//     PlcTask Inputs/G_IO.arDI[75]/Ch[12] <-> Module 1 (GL20-1600END)/1600END input-bit maping/Digital input CH2-bit4
//     PlcTask Inputs/G_IO.arDI[75]/Ch[13] <-> Module 1 (GL20-1600END)/1600END input-bit maping/Digital input CH2-bit5
//     PlcTask Inputs/G_IO.arDI[75]/Ch[14] <-> Module 1 (GL20-1600END)/1600END input-bit maping/Digital input CH2-bit6
//     PlcTask Inputs/G_IO.arDI[75]/Ch[15] <-> Module 1 (GL20-1600END)/1600END input-bit maping/Digital input CH2-bit7
//     PlcTask Inputs/G_IO.arDI[75]/Ch[1] <-> Module 1 (GL20-1600END)/1600END input-bit maping/Digital input CH1-bit1
//     PlcTask Inputs/G_IO.arDI[75]/Ch[2] <-> Module 1 (GL20-1600END)/1600END input-bit maping/Digital input CH1-bit2
//     PlcTask Inputs/G_IO.arDI[75]/Ch[3] <-> Module 1 (GL20-1600END)/1600END input-bit maping/Digital input CH1-bit3
//     PlcTask Inputs/G_IO.arDI[75]/Ch[4] <-> Module 1 (GL20-1600END)/1600END input-bit maping/Digital input CH1-bit4
//     PlcTask Inputs/G_IO.arDI[75]/Ch[5] <-> Module 1 (GL20-1600END)/1600END input-bit maping/Digital input CH1-bit5
//     PlcTask Inputs/G_IO.arDI[75]/Ch[6] <-> Module 1 (GL20-1600END)/1600END input-bit maping/Digital input CH1-bit6
//     PlcTask Inputs/G_IO.arDI[75]/Ch[7] <-> Module 1 (GL20-1600END)/1600END input-bit maping/Digital input CH1-bit7
//     PlcTask Inputs/G_IO.arDI[75]/Ch[8] <-> Module 1 (GL20-1600END)/1600END input-bit maping/Digital input CH2-bit0
//     PlcTask Inputs/G_IO.arDI[75]/Ch[9] <-> Module 1 (GL20-1600END)/1600END input-bit maping/Digital input CH2-bit1
//     PlcTask Outputs/G_IO.arDO[75]/Ch[0] <-> Module 2 (GL20-0016ETP)/0016ETP Output-bit maping/Digital output CH1-bit0
//     PlcTask Outputs/G_IO.arDO[75]/Ch[10] <-> Module 2 (GL20-0016ETP)/0016ETP Output-bit maping/Digital output CH2-bit2
//     PlcTask Outputs/G_IO.arDO[75]/Ch[11] <-> Module 2 (GL20-0016ETP)/0016ETP Output-bit maping/Digital output CH2-bit3
//     PlcTask Outputs/G_IO.arDO[75]/Ch[12] <-> Module 2 (GL20-0016ETP)/0016ETP Output-bit maping/Digital output CH2-bit4
//     PlcTask Outputs/G_IO.arDO[75]/Ch[13] <-> Module 2 (GL20-0016ETP)/0016ETP Output-bit maping/Digital output CH2-bit5
//     PlcTask Outputs/G_IO.arDO[75]/Ch[14] <-> Module 2 (GL20-0016ETP)/0016ETP Output-bit maping/Digital output CH2-bit6
//     PlcTask Outputs/G_IO.arDO[75]/Ch[15] <-> Module 2 (GL20-0016ETP)/0016ETP Output-bit maping/Digital output CH2-bit7
//     PlcTask Outputs/G_IO.arDO[75]/Ch[1] <-> Module 2 (GL20-0016ETP)/0016ETP Output-bit maping/Digital output CH1-bit1
//     PlcTask Outputs/G_IO.arDO[75]/Ch[2] <-> Module 2 (GL20-0016ETP)/0016ETP Output-bit maping/Digital output CH1-bit2
//     PlcTask Outputs/G_IO.arDO[75]/Ch[3] <-> Module 2 (GL20-0016ETP)/0016ETP Output-bit maping/Digital output CH1-bit3
//     PlcTask Outputs/G_IO.arDO[75]/Ch[4] <-> Module 2 (GL20-0016ETP)/0016ETP Output-bit maping/Digital output CH1-bit4
//     PlcTask Outputs/G_IO.arDO[75]/Ch[5] <-> Module 2 (GL20-0016ETP)/0016ETP Output-bit maping/Digital output CH1-bit5
//     PlcTask Outputs/G_IO.arDO[75]/Ch[6] <-> Module 2 (GL20-0016ETP)/0016ETP Output-bit maping/Digital output CH1-bit6
//     PlcTask Outputs/G_IO.arDO[75]/Ch[7] <-> Module 2 (GL20-0016ETP)/0016ETP Output-bit maping/Digital output CH1-bit7
//     PlcTask Outputs/G_IO.arDO[75]/Ch[8] <-> Module 2 (GL20-0016ETP)/0016ETP Output-bit maping/Digital output CH2-bit0
//     PlcTask Outputs/G_IO.arDO[75]/Ch[9] <-> Module 2 (GL20-0016ETP)/0016ETP Output-bit maping/Digital output CH2-bit1
//   kittingDeca/kittingDeca Instance <-> pm side/fr1_dio
//     PlcTask Inputs/G_IO.arDI[76]/Ch[0] <-> Module 1 (GL20-1600END)/1600END input-bit maping/Digital input CH1-bit0
//     PlcTask Inputs/G_IO.arDI[76]/Ch[10] <-> Module 1 (GL20-1600END)/1600END input-bit maping/Digital input CH2-bit2
//     PlcTask Inputs/G_IO.arDI[76]/Ch[11] <-> Module 1 (GL20-1600END)/1600END input-bit maping/Digital input CH2-bit3
//     PlcTask Inputs/G_IO.arDI[76]/Ch[12] <-> Module 1 (GL20-1600END)/1600END input-bit maping/Digital input CH2-bit4
//     PlcTask Inputs/G_IO.arDI[76]/Ch[13] <-> Module 1 (GL20-1600END)/1600END input-bit maping/Digital input CH2-bit5
//     PlcTask Inputs/G_IO.arDI[76]/Ch[14] <-> Module 1 (GL20-1600END)/1600END input-bit maping/Digital input CH2-bit6
//     PlcTask Inputs/G_IO.arDI[76]/Ch[15] <-> Module 1 (GL20-1600END)/1600END input-bit maping/Digital input CH2-bit7
//     PlcTask Inputs/G_IO.arDI[76]/Ch[1] <-> Module 1 (GL20-1600END)/1600END input-bit maping/Digital input CH1-bit1
//     PlcTask Inputs/G_IO.arDI[76]/Ch[2] <-> Module 1 (GL20-1600END)/1600END input-bit maping/Digital input CH1-bit2
//     PlcTask Inputs/G_IO.arDI[76]/Ch[3] <-> Module 1 (GL20-1600END)/1600END input-bit maping/Digital input CH1-bit3
//     PlcTask Inputs/G_IO.arDI[76]/Ch[4] <-> Module 1 (GL20-1600END)/1600END input-bit maping/Digital input CH1-bit4
//     PlcTask Inputs/G_IO.arDI[76]/Ch[5] <-> Module 1 (GL20-1600END)/1600END input-bit maping/Digital input CH1-bit5
//     PlcTask Inputs/G_IO.arDI[76]/Ch[6] <-> Module 1 (GL20-1600END)/1600END input-bit maping/Digital input CH1-bit6
//     PlcTask Inputs/G_IO.arDI[76]/Ch[7] <-> Module 1 (GL20-1600END)/1600END input-bit maping/Digital input CH1-bit7
//     PlcTask Inputs/G_IO.arDI[76]/Ch[8] <-> Module 1 (GL20-1600END)/1600END input-bit maping/Digital input CH2-bit0
//     PlcTask Inputs/G_IO.arDI[76]/Ch[9] <-> Module 1 (GL20-1600END)/1600END input-bit maping/Digital input CH2-bit1
//     PlcTask Outputs/G_IO.arDO[76]/Ch[0] <-> Module 2 (GL20-0016ETP)/0016ETP Output-bit maping/Digital output CH1-bit0
//     PlcTask Outputs/G_IO.arDO[76]/Ch[10] <-> Module 2 (GL20-0016ETP)/0016ETP Output-bit maping/Digital output CH2-bit2
//     PlcTask Outputs/G_IO.arDO[76]/Ch[11] <-> Module 2 (GL20-0016ETP)/0016ETP Output-bit maping/Digital output CH2-bit3
//     PlcTask Outputs/G_IO.arDO[76]/Ch[12] <-> Module 2 (GL20-0016ETP)/0016ETP Output-bit maping/Digital output CH2-bit4
//     PlcTask Outputs/G_IO.arDO[76]/Ch[13] <-> Module 2 (GL20-0016ETP)/0016ETP Output-bit maping/Digital output CH2-bit5
//     PlcTask Outputs/G_IO.arDO[76]/Ch[14] <-> Module 2 (GL20-0016ETP)/0016ETP Output-bit maping/Digital output CH2-bit6
//     PlcTask Outputs/G_IO.arDO[76]/Ch[15] <-> Module 2 (GL20-0016ETP)/0016ETP Output-bit maping/Digital output CH2-bit7
//     PlcTask Outputs/G_IO.arDO[76]/Ch[1] <-> Module 2 (GL20-0016ETP)/0016ETP Output-bit maping/Digital output CH1-bit1
//     PlcTask Outputs/G_IO.arDO[76]/Ch[2] <-> Module 2 (GL20-0016ETP)/0016ETP Output-bit maping/Digital output CH1-bit2
//     PlcTask Outputs/G_IO.arDO[76]/Ch[3] <-> Module 2 (GL20-0016ETP)/0016ETP Output-bit maping/Digital output CH1-bit3
//     PlcTask Outputs/G_IO.arDO[76]/Ch[4] <-> Module 2 (GL20-0016ETP)/0016ETP Output-bit maping/Digital output CH1-bit4
//     PlcTask Outputs/G_IO.arDO[76]/Ch[5] <-> Module 2 (GL20-0016ETP)/0016ETP Output-bit maping/Digital output CH1-bit5
//     PlcTask Outputs/G_IO.arDO[76]/Ch[6] <-> Module 2 (GL20-0016ETP)/0016ETP Output-bit maping/Digital output CH1-bit6
//     PlcTask Outputs/G_IO.arDO[76]/Ch[7] <-> Module 2 (GL20-0016ETP)/0016ETP Output-bit maping/Digital output CH1-bit7
//     PlcTask Outputs/G_IO.arDO[76]/Ch[8] <-> Module 2 (GL20-0016ETP)/0016ETP Output-bit maping/Digital output CH2-bit0
//     PlcTask Outputs/G_IO.arDO[76]/Ch[9] <-> Module 2 (GL20-0016ETP)/0016ETP Output-bit maping/Digital output CH2-bit1
//   kittingDeca/kittingDeca Instance <-> pm side/lb0_converter
//     PlcTask Inputs/GVL.lb[0].belt[0].fbconverter.running_freq <-> Axis#1 Iutputs/Axis1 Running frequency
//     PlcTask Inputs/GVL.lb[0].belt[1].fbconverter.running_freq <-> Axis#2 Iutputs/Axis2 Running frequency
//     PlcTask Inputs/GVL.lb[0].belt[2].fbconverter.running_freq <-> Axis#3 Iutputs/Axis3 Running frequency
//     PlcTask Inputs/GVL.lb[0].belt[0].fbconverter.status <-> Axis#1 Iutputs/Axis1 AC drive running status word 2
//     PlcTask Inputs/GVL.lb[0].belt[1].fbconverter.status <-> Axis#2 Iutputs/Axis2 AC drive running status word 2
//     PlcTask Inputs/GVL.lb[0].belt[2].fbconverter.status <-> Axis#3 Iutputs/Axis3 AC drive running status word 2
//     PlcTask Outputs/GVL.lb[0].belt[0].fbconverter.cmd <-> Axis#1 Outputs/Axis1 Communication control command
//     PlcTask Outputs/GVL.lb[0].belt[1].fbconverter.cmd <-> Axis#2 Outputs/Axis2 Communication control command
//     PlcTask Outputs/GVL.lb[0].belt[2].fbconverter.cmd <-> Axis#3 Outputs/Axis3 Communication control command
//     PlcTask Outputs/GVL.lb[0].belt[0].fbconverter.freq <-> Axis#1 Outputs/Axis1 Frequency set through communication
//     PlcTask Outputs/GVL.lb[0].belt[1].fbconverter.freq <-> Axis#2 Outputs/Axis2 Frequency set through communication
//     PlcTask Outputs/GVL.lb[0].belt[2].fbconverter.freq <-> Axis#3 Outputs/Axis3 Frequency set through communication
//   kittingDeca/kittingDeca Instance <-> pm side/lb0_dio
//     PlcTask Inputs/G_IO.arDI[87]/Ch[0] <-> Module 1 (GL20-1600END)/1600END input-bit maping/Digital input CH1-bit0
//     PlcTask Inputs/G_IO.arDI[87]/Ch[10] <-> Module 1 (GL20-1600END)/1600END input-bit maping/Digital input CH2-bit2
//     PlcTask Inputs/G_IO.arDI[87]/Ch[11] <-> Module 1 (GL20-1600END)/1600END input-bit maping/Digital input CH2-bit3
//     PlcTask Inputs/G_IO.arDI[87]/Ch[12] <-> Module 1 (GL20-1600END)/1600END input-bit maping/Digital input CH2-bit4
//     PlcTask Inputs/G_IO.arDI[87]/Ch[13] <-> Module 1 (GL20-1600END)/1600END input-bit maping/Digital input CH2-bit5
//     PlcTask Inputs/G_IO.arDI[87]/Ch[14] <-> Module 1 (GL20-1600END)/1600END input-bit maping/Digital input CH2-bit6
//     PlcTask Inputs/G_IO.arDI[87]/Ch[15] <-> Module 1 (GL20-1600END)/1600END input-bit maping/Digital input CH2-bit7
//     PlcTask Inputs/G_IO.arDI[87]/Ch[1] <-> Module 1 (GL20-1600END)/1600END input-bit maping/Digital input CH1-bit1
//     PlcTask Inputs/G_IO.arDI[87]/Ch[2] <-> Module 1 (GL20-1600END)/1600END input-bit maping/Digital input CH1-bit2
//     PlcTask Inputs/G_IO.arDI[87]/Ch[3] <-> Module 1 (GL20-1600END)/1600END input-bit maping/Digital input CH1-bit3
//     PlcTask Inputs/G_IO.arDI[87]/Ch[4] <-> Module 1 (GL20-1600END)/1600END input-bit maping/Digital input CH1-bit4
//     PlcTask Inputs/G_IO.arDI[87]/Ch[5] <-> Module 1 (GL20-1600END)/1600END input-bit maping/Digital input CH1-bit5
//     PlcTask Inputs/G_IO.arDI[87]/Ch[6] <-> Module 1 (GL20-1600END)/1600END input-bit maping/Digital input CH1-bit6
//     PlcTask Inputs/G_IO.arDI[87]/Ch[7] <-> Module 1 (GL20-1600END)/1600END input-bit maping/Digital input CH1-bit7
//     PlcTask Inputs/G_IO.arDI[87]/Ch[8] <-> Module 1 (GL20-1600END)/1600END input-bit maping/Digital input CH2-bit0
//     PlcTask Inputs/G_IO.arDI[87]/Ch[9] <-> Module 1 (GL20-1600END)/1600END input-bit maping/Digital input CH2-bit1
//     PlcTask Outputs/G_IO.arDO[87]/Ch[0] <-> Module 2 (GL20-0016ETP)/0016ETP Output-bit maping/Digital output CH1-bit0
//     PlcTask Outputs/G_IO.arDO[87]/Ch[10] <-> Module 2 (GL20-0016ETP)/0016ETP Output-bit maping/Digital output CH2-bit2
//     PlcTask Outputs/G_IO.arDO[87]/Ch[11] <-> Module 2 (GL20-0016ETP)/0016ETP Output-bit maping/Digital output CH2-bit3
//     PlcTask Outputs/G_IO.arDO[87]/Ch[12] <-> Module 2 (GL20-0016ETP)/0016ETP Output-bit maping/Digital output CH2-bit4
//     PlcTask Outputs/G_IO.arDO[87]/Ch[13] <-> Module 2 (GL20-0016ETP)/0016ETP Output-bit maping/Digital output CH2-bit5
//     PlcTask Outputs/G_IO.arDO[87]/Ch[14] <-> Module 2 (GL20-0016ETP)/0016ETP Output-bit maping/Digital output CH2-bit6
//     PlcTask Outputs/G_IO.arDO[87]/Ch[15] <-> Module 2 (GL20-0016ETP)/0016ETP Output-bit maping/Digital output CH2-bit7
//     PlcTask Outputs/G_IO.arDO[87]/Ch[1] <-> Module 2 (GL20-0016ETP)/0016ETP Output-bit maping/Digital output CH1-bit1
//     PlcTask Outputs/G_IO.arDO[87]/Ch[2] <-> Module 2 (GL20-0016ETP)/0016ETP Output-bit maping/Digital output CH1-bit2
//     PlcTask Outputs/G_IO.arDO[87]/Ch[3] <-> Module 2 (GL20-0016ETP)/0016ETP Output-bit maping/Digital output CH1-bit3
//     PlcTask Outputs/G_IO.arDO[87]/Ch[4] <-> Module 2 (GL20-0016ETP)/0016ETP Output-bit maping/Digital output CH1-bit4
//     PlcTask Outputs/G_IO.arDO[87]/Ch[5] <-> Module 2 (GL20-0016ETP)/0016ETP Output-bit maping/Digital output CH1-bit5
//     PlcTask Outputs/G_IO.arDO[87]/Ch[6] <-> Module 2 (GL20-0016ETP)/0016ETP Output-bit maping/Digital output CH1-bit6
//     PlcTask Outputs/G_IO.arDO[87]/Ch[7] <-> Module 2 (GL20-0016ETP)/0016ETP Output-bit maping/Digital output CH1-bit7
//     PlcTask Outputs/G_IO.arDO[87]/Ch[8] <-> Module 2 (GL20-0016ETP)/0016ETP Output-bit maping/Digital output CH2-bit0
//     PlcTask Outputs/G_IO.arDO[87]/Ch[9] <-> Module 2 (GL20-0016ETP)/0016ETP Output-bit maping/Digital output CH2-bit1
//   kittingDeca/kittingDeca Instance <-> pm side/lb1_converter
//     PlcTask Inputs/GVL.lb[1].belt[0].fbconverter.running_freq <-> Axis#1 Iutputs/Axis1 Running frequency
//     PlcTask Inputs/GVL.lb[1].belt[1].fbconverter.running_freq <-> Axis#2 Iutputs/Axis2 Running frequency
//     PlcTask Inputs/GVL.lb[1].belt[2].fbconverter.running_freq <-> Axis#3 Iutputs/Axis3 Running frequency
//     PlcTask Inputs/GVL.lb[1].belt[0].fbconverter.status <-> Axis#1 Iutputs/Axis1 AC drive running status word 2
//     PlcTask Inputs/GVL.lb[1].belt[1].fbconverter.status <-> Axis#2 Iutputs/Axis2 AC drive running status word 2
//     PlcTask Inputs/GVL.lb[1].belt[2].fbconverter.status <-> Axis#3 Iutputs/Axis3 AC drive running status word 2
//     PlcTask Outputs/GVL.lb[1].belt[0].fbconverter.cmd <-> Axis#1 Outputs/Axis1 Communication control command
//     PlcTask Outputs/GVL.lb[1].belt[1].fbconverter.cmd <-> Axis#2 Outputs/Axis2 Communication control command
//     PlcTask Outputs/GVL.lb[1].belt[2].fbconverter.cmd <-> Axis#3 Outputs/Axis3 Communication control command
//     PlcTask Outputs/GVL.lb[1].belt[0].fbconverter.freq <-> Axis#1 Outputs/Axis1 Frequency set through communication
//     PlcTask Outputs/GVL.lb[1].belt[1].fbconverter.freq <-> Axis#2 Outputs/Axis2 Frequency set through communication
//     PlcTask Outputs/GVL.lb[1].belt[2].fbconverter.freq <-> Axis#3 Outputs/Axis3 Frequency set through communication
//   kittingDeca/kittingDeca Instance <-> pm side/lb1_dio
//     PlcTask Inputs/G_IO.arDI[90]/Ch[0] <-> Module 1 (GL20-1600END)/1600END input-bit maping/Digital input CH1-bit0
//     PlcTask Inputs/G_IO.arDI[90]/Ch[10] <-> Module 1 (GL20-1600END)/1600END input-bit maping/Digital input CH2-bit2
//     PlcTask Inputs/G_IO.arDI[90]/Ch[11] <-> Module 1 (GL20-1600END)/1600END input-bit maping/Digital input CH2-bit3
//     PlcTask Inputs/G_IO.arDI[90]/Ch[12] <-> Module 1 (GL20-1600END)/1600END input-bit maping/Digital input CH2-bit4
//     PlcTask Inputs/G_IO.arDI[90]/Ch[13] <-> Module 1 (GL20-1600END)/1600END input-bit maping/Digital input CH2-bit5
//     PlcTask Inputs/G_IO.arDI[90]/Ch[14] <-> Module 1 (GL20-1600END)/1600END input-bit maping/Digital input CH2-bit6
//     PlcTask Inputs/G_IO.arDI[90]/Ch[15] <-> Module 1 (GL20-1600END)/1600END input-bit maping/Digital input CH2-bit7
//     PlcTask Inputs/G_IO.arDI[90]/Ch[1] <-> Module 1 (GL20-1600END)/1600END input-bit maping/Digital input CH1-bit1
//     PlcTask Inputs/G_IO.arDI[90]/Ch[2] <-> Module 1 (GL20-1600END)/1600END input-bit maping/Digital input CH1-bit2
//     PlcTask Inputs/G_IO.arDI[90]/Ch[3] <-> Module 1 (GL20-1600END)/1600END input-bit maping/Digital input CH1-bit3
//     PlcTask Inputs/G_IO.arDI[90]/Ch[4] <-> Module 1 (GL20-1600END)/1600END input-bit maping/Digital input CH1-bit4
//     PlcTask Inputs/G_IO.arDI[90]/Ch[5] <-> Module 1 (GL20-1600END)/1600END input-bit maping/Digital input CH1-bit5
//     PlcTask Inputs/G_IO.arDI[90]/Ch[6] <-> Module 1 (GL20-1600END)/1600END input-bit maping/Digital input CH1-bit6
//     PlcTask Inputs/G_IO.arDI[90]/Ch[7] <-> Module 1 (GL20-1600END)/1600END input-bit maping/Digital input CH1-bit7
//     PlcTask Inputs/G_IO.arDI[90]/Ch[8] <-> Module 1 (GL20-1600END)/1600END input-bit maping/Digital input CH2-bit0
//     PlcTask Inputs/G_IO.arDI[90]/Ch[9] <-> Module 1 (GL20-1600END)/1600END input-bit maping/Digital input CH2-bit1
//     PlcTask Outputs/G_IO.arDO[90]/Ch[0] <-> Module 2 (GL20-0016ETP)/0016ETP Output-bit maping/Digital output CH1-bit0
//     PlcTask Outputs/G_IO.arDO[90]/Ch[10] <-> Module 2 (GL20-0016ETP)/0016ETP Output-bit maping/Digital output CH2-bit2
//     PlcTask Outputs/G_IO.arDO[90]/Ch[11] <-> Module 2 (GL20-0016ETP)/0016ETP Output-bit maping/Digital output CH2-bit3
//     PlcTask Outputs/G_IO.arDO[90]/Ch[12] <-> Module 2 (GL20-0016ETP)/0016ETP Output-bit maping/Digital output CH2-bit4
//     PlcTask Outputs/G_IO.arDO[90]/Ch[13] <-> Module 2 (GL20-0016ETP)/0016ETP Output-bit maping/Digital output CH2-bit5
//     PlcTask Outputs/G_IO.arDO[90]/Ch[14] <-> Module 2 (GL20-0016ETP)/0016ETP Output-bit maping/Digital output CH2-bit6
//     PlcTask Outputs/G_IO.arDO[90]/Ch[15] <-> Module 2 (GL20-0016ETP)/0016ETP Output-bit maping/Digital output CH2-bit7
//     PlcTask Outputs/G_IO.arDO[90]/Ch[1] <-> Module 2 (GL20-0016ETP)/0016ETP Output-bit maping/Digital output CH1-bit1
//     PlcTask Outputs/G_IO.arDO[90]/Ch[2] <-> Module 2 (GL20-0016ETP)/0016ETP Output-bit maping/Digital output CH1-bit2
//     PlcTask Outputs/G_IO.arDO[90]/Ch[3] <-> Module 2 (GL20-0016ETP)/0016ETP Output-bit maping/Digital output CH1-bit3
//     PlcTask Outputs/G_IO.arDO[90]/Ch[4] <-> Module 2 (GL20-0016ETP)/0016ETP Output-bit maping/Digital output CH1-bit4
//     PlcTask Outputs/G_IO.arDO[90]/Ch[5] <-> Module 2 (GL20-0016ETP)/0016ETP Output-bit maping/Digital output CH1-bit5
//     PlcTask Outputs/G_IO.arDO[90]/Ch[6] <-> Module 2 (GL20-0016ETP)/0016ETP Output-bit maping/Digital output CH1-bit6
//     PlcTask Outputs/G_IO.arDO[90]/Ch[7] <-> Module 2 (GL20-0016ETP)/0016ETP Output-bit maping/Digital output CH1-bit7
//     PlcTask Outputs/G_IO.arDO[90]/Ch[8] <-> Module 2 (GL20-0016ETP)/0016ETP Output-bit maping/Digital output CH2-bit0
//     PlcTask Outputs/G_IO.arDO[90]/Ch[9] <-> Module 2 (GL20-0016ETP)/0016ETP Output-bit maping/Digital output CH2-bit1
//   kittingDeca/kittingDeca Instance <-> pm side/lc0_converter
//     PlcTask Inputs/GVL.lc[0].belt_out.belt.fbconverter.running_freq <-> Axis#1 Iutputs/Axis1 Running frequency
//     PlcTask Inputs/GVL.lc[0].belt_out.belt.fbconverter.status <-> Axis#1 Iutputs/Axis1 AC drive running status word 2
//     PlcTask Outputs/GVL.lc[0].belt_out.belt.fbconverter.cmd <-> Axis#1 Outputs/Axis1 Communication control command
//     PlcTask Outputs/GVL.lc[0].belt_out.belt.fbconverter.freq <-> Axis#1 Outputs/Axis1 Frequency set through communication
//   kittingDeca/kittingDeca Instance <-> pm side/lc0_dio
//     PlcTask Inputs/G_IO.arDI[85]/Ch[0] <-> Module 1 (GL20-1600END)/1600END input-bit maping/Digital input CH1-bit0
//     PlcTask Inputs/G_IO.arDI[85]/Ch[10] <-> Module 1 (GL20-1600END)/1600END input-bit maping/Digital input CH2-bit2
//     PlcTask Inputs/G_IO.arDI[85]/Ch[11] <-> Module 1 (GL20-1600END)/1600END input-bit maping/Digital input CH2-bit3
//     PlcTask Inputs/G_IO.arDI[85]/Ch[12] <-> Module 1 (GL20-1600END)/1600END input-bit maping/Digital input CH2-bit4
//     PlcTask Inputs/G_IO.arDI[85]/Ch[13] <-> Module 1 (GL20-1600END)/1600END input-bit maping/Digital input CH2-bit5
//     PlcTask Inputs/G_IO.arDI[85]/Ch[14] <-> Module 1 (GL20-1600END)/1600END input-bit maping/Digital input CH2-bit6
//     PlcTask Inputs/G_IO.arDI[85]/Ch[15] <-> Module 1 (GL20-1600END)/1600END input-bit maping/Digital input CH2-bit7
//     PlcTask Inputs/G_IO.arDI[85]/Ch[1] <-> Module 1 (GL20-1600END)/1600END input-bit maping/Digital input CH1-bit1
//     PlcTask Inputs/G_IO.arDI[85]/Ch[2] <-> Module 1 (GL20-1600END)/1600END input-bit maping/Digital input CH1-bit2
//     PlcTask Inputs/G_IO.arDI[85]/Ch[3] <-> Module 1 (GL20-1600END)/1600END input-bit maping/Digital input CH1-bit3
//     PlcTask Inputs/G_IO.arDI[85]/Ch[4] <-> Module 1 (GL20-1600END)/1600END input-bit maping/Digital input CH1-bit4
//     PlcTask Inputs/G_IO.arDI[85]/Ch[5] <-> Module 1 (GL20-1600END)/1600END input-bit maping/Digital input CH1-bit5
//     PlcTask Inputs/G_IO.arDI[85]/Ch[6] <-> Module 1 (GL20-1600END)/1600END input-bit maping/Digital input CH1-bit6
//     PlcTask Inputs/G_IO.arDI[85]/Ch[7] <-> Module 1 (GL20-1600END)/1600END input-bit maping/Digital input CH1-bit7
//     PlcTask Inputs/G_IO.arDI[85]/Ch[8] <-> Module 1 (GL20-1600END)/1600END input-bit maping/Digital input CH2-bit0
//     PlcTask Inputs/G_IO.arDI[85]/Ch[9] <-> Module 1 (GL20-1600END)/1600END input-bit maping/Digital input CH2-bit1
//     PlcTask Inputs/G_IO.arDI[86]/Ch[0] <-> Module 2 (GL20-1600END)/1600END input-bit maping/Digital input CH1-bit0
//     PlcTask Inputs/G_IO.arDI[86]/Ch[10] <-> Module 2 (GL20-1600END)/1600END input-bit maping/Digital input CH2-bit2
//     PlcTask Inputs/G_IO.arDI[86]/Ch[11] <-> Module 2 (GL20-1600END)/1600END input-bit maping/Digital input CH2-bit3
//     PlcTask Inputs/G_IO.arDI[86]/Ch[12] <-> Module 2 (GL20-1600END)/1600END input-bit maping/Digital input CH2-bit4
//     PlcTask Inputs/G_IO.arDI[86]/Ch[13] <-> Module 2 (GL20-1600END)/1600END input-bit maping/Digital input CH2-bit5
//     PlcTask Inputs/G_IO.arDI[86]/Ch[14] <-> Module 2 (GL20-1600END)/1600END input-bit maping/Digital input CH2-bit6
//     PlcTask Inputs/G_IO.arDI[86]/Ch[15] <-> Module 2 (GL20-1600END)/1600END input-bit maping/Digital input CH2-bit7
//     PlcTask Inputs/G_IO.arDI[86]/Ch[1] <-> Module 2 (GL20-1600END)/1600END input-bit maping/Digital input CH1-bit1
//     PlcTask Inputs/G_IO.arDI[86]/Ch[2] <-> Module 2 (GL20-1600END)/1600END input-bit maping/Digital input CH1-bit2
//     PlcTask Inputs/G_IO.arDI[86]/Ch[3] <-> Module 2 (GL20-1600END)/1600END input-bit maping/Digital input CH1-bit3
//     PlcTask Inputs/G_IO.arDI[86]/Ch[4] <-> Module 2 (GL20-1600END)/1600END input-bit maping/Digital input CH1-bit4
//     PlcTask Inputs/G_IO.arDI[86]/Ch[5] <-> Module 2 (GL20-1600END)/1600END input-bit maping/Digital input CH1-bit5
//     PlcTask Inputs/G_IO.arDI[86]/Ch[6] <-> Module 2 (GL20-1600END)/1600END input-bit maping/Digital input CH1-bit6
//     PlcTask Inputs/G_IO.arDI[86]/Ch[7] <-> Module 2 (GL20-1600END)/1600END input-bit maping/Digital input CH1-bit7
//     PlcTask Inputs/G_IO.arDI[86]/Ch[8] <-> Module 2 (GL20-1600END)/1600END input-bit maping/Digital input CH2-bit0
//     PlcTask Inputs/G_IO.arDI[86]/Ch[9] <-> Module 2 (GL20-1600END)/1600END input-bit maping/Digital input CH2-bit1
//     PlcTask Outputs/G_IO.arDO[85]/Ch[0] <-> Module 3 (GL20-0016ETP)/0016ETP Output-bit maping/Digital output CH1-bit0
//     PlcTask Outputs/G_IO.arDO[85]/Ch[10] <-> Module 3 (GL20-0016ETP)/0016ETP Output-bit maping/Digital output CH2-bit2
//     PlcTask Outputs/G_IO.arDO[85]/Ch[11] <-> Module 3 (GL20-0016ETP)/0016ETP Output-bit maping/Digital output CH2-bit3
//     PlcTask Outputs/G_IO.arDO[85]/Ch[12] <-> Module 3 (GL20-0016ETP)/0016ETP Output-bit maping/Digital output CH2-bit4
//     PlcTask Outputs/G_IO.arDO[85]/Ch[13] <-> Module 3 (GL20-0016ETP)/0016ETP Output-bit maping/Digital output CH2-bit5
//     PlcTask Outputs/G_IO.arDO[85]/Ch[14] <-> Module 3 (GL20-0016ETP)/0016ETP Output-bit maping/Digital output CH2-bit6
//     PlcTask Outputs/G_IO.arDO[85]/Ch[15] <-> Module 3 (GL20-0016ETP)/0016ETP Output-bit maping/Digital output CH2-bit7
//     PlcTask Outputs/G_IO.arDO[85]/Ch[1] <-> Module 3 (GL20-0016ETP)/0016ETP Output-bit maping/Digital output CH1-bit1
//     PlcTask Outputs/G_IO.arDO[85]/Ch[2] <-> Module 3 (GL20-0016ETP)/0016ETP Output-bit maping/Digital output CH1-bit2
//     PlcTask Outputs/G_IO.arDO[85]/Ch[3] <-> Module 3 (GL20-0016ETP)/0016ETP Output-bit maping/Digital output CH1-bit3
//     PlcTask Outputs/G_IO.arDO[85]/Ch[4] <-> Module 3 (GL20-0016ETP)/0016ETP Output-bit maping/Digital output CH1-bit4
//     PlcTask Outputs/G_IO.arDO[85]/Ch[5] <-> Module 3 (GL20-0016ETP)/0016ETP Output-bit maping/Digital output CH1-bit5
//     PlcTask Outputs/G_IO.arDO[85]/Ch[6] <-> Module 3 (GL20-0016ETP)/0016ETP Output-bit maping/Digital output CH1-bit6
//     PlcTask Outputs/G_IO.arDO[85]/Ch[7] <-> Module 3 (GL20-0016ETP)/0016ETP Output-bit maping/Digital output CH1-bit7
//     PlcTask Outputs/G_IO.arDO[85]/Ch[8] <-> Module 3 (GL20-0016ETP)/0016ETP Output-bit maping/Digital output CH2-bit0
//     PlcTask Outputs/G_IO.arDO[85]/Ch[9] <-> Module 3 (GL20-0016ETP)/0016ETP Output-bit maping/Digital output CH2-bit1
//     PlcTask Outputs/G_IO.arDO[86]/Ch[0] <-> Module 4 (GL20-0016ETP)/0016ETP Output-bit maping/Digital output CH1-bit0
//     PlcTask Outputs/G_IO.arDO[86]/Ch[10] <-> Module 4 (GL20-0016ETP)/0016ETP Output-bit maping/Digital output CH2-bit2
//     PlcTask Outputs/G_IO.arDO[86]/Ch[11] <-> Module 4 (GL20-0016ETP)/0016ETP Output-bit maping/Digital output CH2-bit3
//     PlcTask Outputs/G_IO.arDO[86]/Ch[12] <-> Module 4 (GL20-0016ETP)/0016ETP Output-bit maping/Digital output CH2-bit4
//     PlcTask Outputs/G_IO.arDO[86]/Ch[13] <-> Module 4 (GL20-0016ETP)/0016ETP Output-bit maping/Digital output CH2-bit5
//     PlcTask Outputs/G_IO.arDO[86]/Ch[14] <-> Module 4 (GL20-0016ETP)/0016ETP Output-bit maping/Digital output CH2-bit6
//     PlcTask Outputs/G_IO.arDO[86]/Ch[15] <-> Module 4 (GL20-0016ETP)/0016ETP Output-bit maping/Digital output CH2-bit7
//     PlcTask Outputs/G_IO.arDO[86]/Ch[1] <-> Module 4 (GL20-0016ETP)/0016ETP Output-bit maping/Digital output CH1-bit1
//     PlcTask Outputs/G_IO.arDO[86]/Ch[2] <-> Module 4 (GL20-0016ETP)/0016ETP Output-bit maping/Digital output CH1-bit2
//     PlcTask Outputs/G_IO.arDO[86]/Ch[3] <-> Module 4 (GL20-0016ETP)/0016ETP Output-bit maping/Digital output CH1-bit3
//     PlcTask Outputs/G_IO.arDO[86]/Ch[4] <-> Module 4 (GL20-0016ETP)/0016ETP Output-bit maping/Digital output CH1-bit4
//     PlcTask Outputs/G_IO.arDO[86]/Ch[5] <-> Module 4 (GL20-0016ETP)/0016ETP Output-bit maping/Digital output CH1-bit5
//     PlcTask Outputs/G_IO.arDO[86]/Ch[6] <-> Module 4 (GL20-0016ETP)/0016ETP Output-bit maping/Digital output CH1-bit6
//     PlcTask Outputs/G_IO.arDO[86]/Ch[7] <-> Module 4 (GL20-0016ETP)/0016ETP Output-bit maping/Digital output CH1-bit7
//     PlcTask Outputs/G_IO.arDO[86]/Ch[8] <-> Module 4 (GL20-0016ETP)/0016ETP Output-bit maping/Digital output CH2-bit0
//     PlcTask Outputs/G_IO.arDO[86]/Ch[9] <-> Module 4 (GL20-0016ETP)/0016ETP Output-bit maping/Digital output CH2-bit1
//   kittingDeca/kittingDeca Instance <-> pm side/lc1_converter
//     PlcTask Inputs/GVL.lc[1].belt_out.belt.fbconverter.running_freq <-> Axis#1 Iutputs/Axis1 Running frequency
//     PlcTask Inputs/GVL.lc[1].belt_out.belt.fbconverter.status <-> Axis#1 Iutputs/Axis1 AC drive running status word 2
//     PlcTask Outputs/GVL.lc[1].belt_out.belt.fbconverter.cmd <-> Axis#1 Outputs/Axis1 Communication control command
//     PlcTask Outputs/GVL.lc[1].belt_out.belt.fbconverter.freq <-> Axis#1 Outputs/Axis1 Frequency set through communication
//   kittingDeca/kittingDeca Instance <-> pm side/lc1_dio
//     PlcTask Inputs/G_IO.arDI[88]/Ch[0] <-> Module 1 (GL20-1600END)/1600END input-bit maping/Digital input CH1-bit0
//     PlcTask Inputs/G_IO.arDI[88]/Ch[10] <-> Module 1 (GL20-1600END)/1600END input-bit maping/Digital input CH2-bit2
//     PlcTask Inputs/G_IO.arDI[88]/Ch[11] <-> Module 1 (GL20-1600END)/1600END input-bit maping/Digital input CH2-bit3
//     PlcTask Inputs/G_IO.arDI[88]/Ch[12] <-> Module 1 (GL20-1600END)/1600END input-bit maping/Digital input CH2-bit4
//     PlcTask Inputs/G_IO.arDI[88]/Ch[13] <-> Module 1 (GL20-1600END)/1600END input-bit maping/Digital input CH2-bit5
//     PlcTask Inputs/G_IO.arDI[88]/Ch[14] <-> Module 1 (GL20-1600END)/1600END input-bit maping/Digital input CH2-bit6
//     PlcTask Inputs/G_IO.arDI[88]/Ch[15] <-> Module 1 (GL20-1600END)/1600END input-bit maping/Digital input CH2-bit7
//     PlcTask Inputs/G_IO.arDI[88]/Ch[1] <-> Module 1 (GL20-1600END)/1600END input-bit maping/Digital input CH1-bit1
//     PlcTask Inputs/G_IO.arDI[88]/Ch[2] <-> Module 1 (GL20-1600END)/1600END input-bit maping/Digital input CH1-bit2
//     PlcTask Inputs/G_IO.arDI[88]/Ch[3] <-> Module 1 (GL20-1600END)/1600END input-bit maping/Digital input CH1-bit3
//     PlcTask Inputs/G_IO.arDI[88]/Ch[4] <-> Module 1 (GL20-1600END)/1600END input-bit maping/Digital input CH1-bit4
//     PlcTask Inputs/G_IO.arDI[88]/Ch[5] <-> Module 1 (GL20-1600END)/1600END input-bit maping/Digital input CH1-bit5
//     PlcTask Inputs/G_IO.arDI[88]/Ch[6] <-> Module 1 (GL20-1600END)/1600END input-bit maping/Digital input CH1-bit6
//     PlcTask Inputs/G_IO.arDI[88]/Ch[7] <-> Module 1 (GL20-1600END)/1600END input-bit maping/Digital input CH1-bit7
//     PlcTask Inputs/G_IO.arDI[88]/Ch[8] <-> Module 1 (GL20-1600END)/1600END input-bit maping/Digital input CH2-bit0
//     PlcTask Inputs/G_IO.arDI[88]/Ch[9] <-> Module 1 (GL20-1600END)/1600END input-bit maping/Digital input CH2-bit1
//     PlcTask Inputs/G_IO.arDI[89]/Ch[0] <-> Module 2 (GL20-1600END)/1600END input-bit maping/Digital input CH1-bit0
//     PlcTask Inputs/G_IO.arDI[89]/Ch[10] <-> Module 2 (GL20-1600END)/1600END input-bit maping/Digital input CH2-bit2
//     PlcTask Inputs/G_IO.arDI[89]/Ch[11] <-> Module 2 (GL20-1600END)/1600END input-bit maping/Digital input CH2-bit3
//     PlcTask Inputs/G_IO.arDI[89]/Ch[12] <-> Module 2 (GL20-1600END)/1600END input-bit maping/Digital input CH2-bit4
//     PlcTask Inputs/G_IO.arDI[89]/Ch[13] <-> Module 2 (GL20-1600END)/1600END input-bit maping/Digital input CH2-bit5
//     PlcTask Inputs/G_IO.arDI[89]/Ch[14] <-> Module 2 (GL20-1600END)/1600END input-bit maping/Digital input CH2-bit6
//     PlcTask Inputs/G_IO.arDI[89]/Ch[15] <-> Module 2 (GL20-1600END)/1600END input-bit maping/Digital input CH2-bit7
//     PlcTask Inputs/G_IO.arDI[89]/Ch[1] <-> Module 2 (GL20-1600END)/1600END input-bit maping/Digital input CH1-bit1
//     PlcTask Inputs/G_IO.arDI[89]/Ch[2] <-> Module 2 (GL20-1600END)/1600END input-bit maping/Digital input CH1-bit2
//     PlcTask Inputs/G_IO.arDI[89]/Ch[3] <-> Module 2 (GL20-1600END)/1600END input-bit maping/Digital input CH1-bit3
//     PlcTask Inputs/G_IO.arDI[89]/Ch[4] <-> Module 2 (GL20-1600END)/1600END input-bit maping/Digital input CH1-bit4
//     PlcTask Inputs/G_IO.arDI[89]/Ch[5] <-> Module 2 (GL20-1600END)/1600END input-bit maping/Digital input CH1-bit5
//     PlcTask Inputs/G_IO.arDI[89]/Ch[6] <-> Module 2 (GL20-1600END)/1600END input-bit maping/Digital input CH1-bit6
//     PlcTask Inputs/G_IO.arDI[89]/Ch[7] <-> Module 2 (GL20-1600END)/1600END input-bit maping/Digital input CH1-bit7
//     PlcTask Inputs/G_IO.arDI[89]/Ch[8] <-> Module 2 (GL20-1600END)/1600END input-bit maping/Digital input CH2-bit0
//     PlcTask Inputs/G_IO.arDI[89]/Ch[9] <-> Module 2 (GL20-1600END)/1600END input-bit maping/Digital input CH2-bit1
//     PlcTask Outputs/G_IO.arDO[88]/Ch[0] <-> Module 3 (GL20-0016ETP)/0016ETP Output-bit maping/Digital output CH1-bit0
//     PlcTask Outputs/G_IO.arDO[88]/Ch[10] <-> Module 3 (GL20-0016ETP)/0016ETP Output-bit maping/Digital output CH2-bit2
//     PlcTask Outputs/G_IO.arDO[88]/Ch[11] <-> Module 3 (GL20-0016ETP)/0016ETP Output-bit maping/Digital output CH2-bit3
//     PlcTask Outputs/G_IO.arDO[88]/Ch[12] <-> Module 3 (GL20-0016ETP)/0016ETP Output-bit maping/Digital output CH2-bit4
//     PlcTask Outputs/G_IO.arDO[88]/Ch[13] <-> Module 3 (GL20-0016ETP)/0016ETP Output-bit maping/Digital output CH2-bit5
//     PlcTask Outputs/G_IO.arDO[88]/Ch[14] <-> Module 3 (GL20-0016ETP)/0016ETP Output-bit maping/Digital output CH2-bit6
//     PlcTask Outputs/G_IO.arDO[88]/Ch[15] <-> Module 3 (GL20-0016ETP)/0016ETP Output-bit maping/Digital output CH2-bit7
//     PlcTask Outputs/G_IO.arDO[88]/Ch[1] <-> Module 3 (GL20-0016ETP)/0016ETP Output-bit maping/Digital output CH1-bit1
//     PlcTask Outputs/G_IO.arDO[88]/Ch[2] <-> Module 3 (GL20-0016ETP)/0016ETP Output-bit maping/Digital output CH1-bit2
//     PlcTask Outputs/G_IO.arDO[88]/Ch[3] <-> Module 3 (GL20-0016ETP)/0016ETP Output-bit maping/Digital output CH1-bit3
//     PlcTask Outputs/G_IO.arDO[88]/Ch[4] <-> Module 3 (GL20-0016ETP)/0016ETP Output-bit maping/Digital output CH1-bit4
//     PlcTask Outputs/G_IO.arDO[88]/Ch[5] <-> Module 3 (GL20-0016ETP)/0016ETP Output-bit maping/Digital output CH1-bit5
//     PlcTask Outputs/G_IO.arDO[88]/Ch[6] <-> Module 3 (GL20-0016ETP)/0016ETP Output-bit maping/Digital output CH1-bit6
//     PlcTask Outputs/G_IO.arDO[88]/Ch[7] <-> Module 3 (GL20-0016ETP)/0016ETP Output-bit maping/Digital output CH1-bit7
//     PlcTask Outputs/G_IO.arDO[88]/Ch[8] <-> Module 3 (GL20-0016ETP)/0016ETP Output-bit maping/Digital output CH2-bit0
//     PlcTask Outputs/G_IO.arDO[88]/Ch[9] <-> Module 3 (GL20-0016ETP)/0016ETP Output-bit maping/Digital output CH2-bit1
//     PlcTask Outputs/G_IO.arDO[89]/Ch[0] <-> Module 4 (GL20-0016ETP)/0016ETP Output-bit maping/Digital output CH1-bit0
//     PlcTask Outputs/G_IO.arDO[89]/Ch[10] <-> Module 4 (GL20-0016ETP)/0016ETP Output-bit maping/Digital output CH2-bit2
//     PlcTask Outputs/G_IO.arDO[89]/Ch[11] <-> Module 4 (GL20-0016ETP)/0016ETP Output-bit maping/Digital output CH2-bit3
//     PlcTask Outputs/G_IO.arDO[89]/Ch[12] <-> Module 4 (GL20-0016ETP)/0016ETP Output-bit maping/Digital output CH2-bit4
//     PlcTask Outputs/G_IO.arDO[89]/Ch[13] <-> Module 4 (GL20-0016ETP)/0016ETP Output-bit maping/Digital output CH2-bit5
//     PlcTask Outputs/G_IO.arDO[89]/Ch[14] <-> Module 4 (GL20-0016ETP)/0016ETP Output-bit maping/Digital output CH2-bit6
//     PlcTask Outputs/G_IO.arDO[89]/Ch[15] <-> Module 4 (GL20-0016ETP)/0016ETP Output-bit maping/Digital output CH2-bit7
//     PlcTask Outputs/G_IO.arDO[89]/Ch[1] <-> Module 4 (GL20-0016ETP)/0016ETP Output-bit maping/Digital output CH1-bit1
//     PlcTask Outputs/G_IO.arDO[89]/Ch[2] <-> Module 4 (GL20-0016ETP)/0016ETP Output-bit maping/Digital output CH1-bit2
//     PlcTask Outputs/G_IO.arDO[89]/Ch[3] <-> Module 4 (GL20-0016ETP)/0016ETP Output-bit maping/Digital output CH1-bit3
//     PlcTask Outputs/G_IO.arDO[89]/Ch[4] <-> Module 4 (GL20-0016ETP)/0016ETP Output-bit maping/Digital output CH1-bit4
//     PlcTask Outputs/G_IO.arDO[89]/Ch[5] <-> Module 4 (GL20-0016ETP)/0016ETP Output-bit maping/Digital output CH1-bit5
//     PlcTask Outputs/G_IO.arDO[89]/Ch[6] <-> Module 4 (GL20-0016ETP)/0016ETP Output-bit maping/Digital output CH1-bit6
//     PlcTask Outputs/G_IO.arDO[89]/Ch[7] <-> Module 4 (GL20-0016ETP)/0016ETP Output-bit maping/Digital output CH1-bit7
//     PlcTask Outputs/G_IO.arDO[89]/Ch[8] <-> Module 4 (GL20-0016ETP)/0016ETP Output-bit maping/Digital output CH2-bit0
//     PlcTask Outputs/G_IO.arDO[89]/Ch[9] <-> Module 4 (GL20-0016ETP)/0016ETP Output-bit maping/Digital output CH2-bit1
//   kittingDeca/kittingDeca Instance <-> pm side/pm0_1_dio
//     PlcTask Inputs/G_IO.arDI[50]/Ch[0] <-> Module 1 (GL20-1600END)/1600END input-bit maping/Digital input CH1-bit0
//     PlcTask Inputs/G_IO.arDI[50]/Ch[10] <-> Module 1 (GL20-1600END)/1600END input-bit maping/Digital input CH2-bit2
//     PlcTask Inputs/G_IO.arDI[50]/Ch[11] <-> Module 1 (GL20-1600END)/1600END input-bit maping/Digital input CH2-bit3
//     PlcTask Inputs/G_IO.arDI[50]/Ch[12] <-> Module 1 (GL20-1600END)/1600END input-bit maping/Digital input CH2-bit4
//     PlcTask Inputs/G_IO.arDI[50]/Ch[13] <-> Module 1 (GL20-1600END)/1600END input-bit maping/Digital input CH2-bit5
//     PlcTask Inputs/G_IO.arDI[50]/Ch[14] <-> Module 1 (GL20-1600END)/1600END input-bit maping/Digital input CH2-bit6
//     PlcTask Inputs/G_IO.arDI[50]/Ch[15] <-> Module 1 (GL20-1600END)/1600END input-bit maping/Digital input CH2-bit7
//     PlcTask Inputs/G_IO.arDI[50]/Ch[1] <-> Module 1 (GL20-1600END)/1600END input-bit maping/Digital input CH1-bit1
//     PlcTask Inputs/G_IO.arDI[50]/Ch[2] <-> Module 1 (GL20-1600END)/1600END input-bit maping/Digital input CH1-bit2
//     PlcTask Inputs/G_IO.arDI[50]/Ch[3] <-> Module 1 (GL20-1600END)/1600END input-bit maping/Digital input CH1-bit3
//     PlcTask Inputs/G_IO.arDI[50]/Ch[4] <-> Module 1 (GL20-1600END)/1600END input-bit maping/Digital input CH1-bit4
//     PlcTask Inputs/G_IO.arDI[50]/Ch[5] <-> Module 1 (GL20-1600END)/1600END input-bit maping/Digital input CH1-bit5
//     PlcTask Inputs/G_IO.arDI[50]/Ch[6] <-> Module 1 (GL20-1600END)/1600END input-bit maping/Digital input CH1-bit6
//     PlcTask Inputs/G_IO.arDI[50]/Ch[7] <-> Module 1 (GL20-1600END)/1600END input-bit maping/Digital input CH1-bit7
//     PlcTask Inputs/G_IO.arDI[50]/Ch[8] <-> Module 1 (GL20-1600END)/1600END input-bit maping/Digital input CH2-bit0
//     PlcTask Inputs/G_IO.arDI[50]/Ch[9] <-> Module 1 (GL20-1600END)/1600END input-bit maping/Digital input CH2-bit1
//     PlcTask Inputs/G_IO.arDI[51]/Ch[0] <-> Module 2 (GL20-1600END)/1600END input-bit maping/Digital input CH1-bit0
//     PlcTask Inputs/G_IO.arDI[51]/Ch[10] <-> Module 2 (GL20-1600END)/1600END input-bit maping/Digital input CH2-bit2
//     PlcTask Inputs/G_IO.arDI[51]/Ch[11] <-> Module 2 (GL20-1600END)/1600END input-bit maping/Digital input CH2-bit3
//     PlcTask Inputs/G_IO.arDI[51]/Ch[12] <-> Module 2 (GL20-1600END)/1600END input-bit maping/Digital input CH2-bit4
//     PlcTask Inputs/G_IO.arDI[51]/Ch[13] <-> Module 2 (GL20-1600END)/1600END input-bit maping/Digital input CH2-bit5
//     PlcTask Inputs/G_IO.arDI[51]/Ch[14] <-> Module 2 (GL20-1600END)/1600END input-bit maping/Digital input CH2-bit6
//     PlcTask Inputs/G_IO.arDI[51]/Ch[15] <-> Module 2 (GL20-1600END)/1600END input-bit maping/Digital input CH2-bit7
//     PlcTask Inputs/G_IO.arDI[51]/Ch[1] <-> Module 2 (GL20-1600END)/1600END input-bit maping/Digital input CH1-bit1
//     PlcTask Inputs/G_IO.arDI[51]/Ch[2] <-> Module 2 (GL20-1600END)/1600END input-bit maping/Digital input CH1-bit2
//     PlcTask Inputs/G_IO.arDI[51]/Ch[3] <-> Module 2 (GL20-1600END)/1600END input-bit maping/Digital input CH1-bit3
//     PlcTask Inputs/G_IO.arDI[51]/Ch[4] <-> Module 2 (GL20-1600END)/1600END input-bit maping/Digital input CH1-bit4
//     PlcTask Inputs/G_IO.arDI[51]/Ch[5] <-> Module 2 (GL20-1600END)/1600END input-bit maping/Digital input CH1-bit5
//     PlcTask Inputs/G_IO.arDI[51]/Ch[6] <-> Module 2 (GL20-1600END)/1600END input-bit maping/Digital input CH1-bit6
//     PlcTask Inputs/G_IO.arDI[51]/Ch[7] <-> Module 2 (GL20-1600END)/1600END input-bit maping/Digital input CH1-bit7
//     PlcTask Inputs/G_IO.arDI[51]/Ch[8] <-> Module 2 (GL20-1600END)/1600END input-bit maping/Digital input CH2-bit0
//     PlcTask Inputs/G_IO.arDI[51]/Ch[9] <-> Module 2 (GL20-1600END)/1600END input-bit maping/Digital input CH2-bit1
//     PlcTask Inputs/G_IO.arDI[52]/Ch[0] <-> Module 3 (GL20-1600END)/1600END input-bit maping/Digital input CH1-bit0
//     PlcTask Inputs/G_IO.arDI[52]/Ch[10] <-> Module 3 (GL20-1600END)/1600END input-bit maping/Digital input CH2-bit2
//     PlcTask Inputs/G_IO.arDI[52]/Ch[11] <-> Module 3 (GL20-1600END)/1600END input-bit maping/Digital input CH2-bit3
//     PlcTask Inputs/G_IO.arDI[52]/Ch[12] <-> Module 3 (GL20-1600END)/1600END input-bit maping/Digital input CH2-bit4
//     PlcTask Inputs/G_IO.arDI[52]/Ch[13] <-> Module 3 (GL20-1600END)/1600END input-bit maping/Digital input CH2-bit5
//     PlcTask Inputs/G_IO.arDI[52]/Ch[14] <-> Module 3 (GL20-1600END)/1600END input-bit maping/Digital input CH2-bit6
//     PlcTask Inputs/G_IO.arDI[52]/Ch[15] <-> Module 3 (GL20-1600END)/1600END input-bit maping/Digital input CH2-bit7
//     PlcTask Inputs/G_IO.arDI[52]/Ch[1] <-> Module 3 (GL20-1600END)/1600END input-bit maping/Digital input CH1-bit1
//     PlcTask Inputs/G_IO.arDI[52]/Ch[2] <-> Module 3 (GL20-1600END)/1600END input-bit maping/Digital input CH1-bit2
//     PlcTask Inputs/G_IO.arDI[52]/Ch[3] <-> Module 3 (GL20-1600END)/1600END input-bit maping/Digital input CH1-bit3
//     PlcTask Inputs/G_IO.arDI[52]/Ch[4] <-> Module 3 (GL20-1600END)/1600END input-bit maping/Digital input CH1-bit4
//     PlcTask Inputs/G_IO.arDI[52]/Ch[5] <-> Module 3 (GL20-1600END)/1600END input-bit maping/Digital input CH1-bit5
//     PlcTask Inputs/G_IO.arDI[52]/Ch[6] <-> Module 3 (GL20-1600END)/1600END input-bit maping/Digital input CH1-bit6
//     PlcTask Inputs/G_IO.arDI[52]/Ch[7] <-> Module 3 (GL20-1600END)/1600END input-bit maping/Digital input CH1-bit7
//     PlcTask Inputs/G_IO.arDI[52]/Ch[8] <-> Module 3 (GL20-1600END)/1600END input-bit maping/Digital input CH2-bit0
//     PlcTask Inputs/G_IO.arDI[52]/Ch[9] <-> Module 3 (GL20-1600END)/1600END input-bit maping/Digital input CH2-bit1
//     PlcTask Inputs/G_IO.arDI[53]/Ch[0] <-> Module 4 (GL20-1600END)/1600END input-bit maping/Digital input CH1-bit0
//     PlcTask Inputs/G_IO.arDI[53]/Ch[10] <-> Module 4 (GL20-1600END)/1600END input-bit maping/Digital input CH2-bit2
//     PlcTask Inputs/G_IO.arDI[53]/Ch[11] <-> Module 4 (GL20-1600END)/1600END input-bit maping/Digital input CH2-bit3
//     PlcTask Inputs/G_IO.arDI[53]/Ch[12] <-> Module 4 (GL20-1600END)/1600END input-bit maping/Digital input CH2-bit4
//     PlcTask Inputs/G_IO.arDI[53]/Ch[13] <-> Module 4 (GL20-1600END)/1600END input-bit maping/Digital input CH2-bit5
//     PlcTask Inputs/G_IO.arDI[53]/Ch[14] <-> Module 4 (GL20-1600END)/1600END input-bit maping/Digital input CH2-bit6
//     PlcTask Inputs/G_IO.arDI[53]/Ch[15] <-> Module 4 (GL20-1600END)/1600END input-bit maping/Digital input CH2-bit7
//     PlcTask Inputs/G_IO.arDI[53]/Ch[1] <-> Module 4 (GL20-1600END)/1600END input-bit maping/Digital input CH1-bit1
//     PlcTask Inputs/G_IO.arDI[53]/Ch[2] <-> Module 4 (GL20-1600END)/1600END input-bit maping/Digital input CH1-bit2
//     PlcTask Inputs/G_IO.arDI[53]/Ch[3] <-> Module 4 (GL20-1600END)/1600END input-bit maping/Digital input CH1-bit3
//     PlcTask Inputs/G_IO.arDI[53]/Ch[4] <-> Module 4 (GL20-1600END)/1600END input-bit maping/Digital input CH1-bit4
//     PlcTask Inputs/G_IO.arDI[53]/Ch[5] <-> Module 4 (GL20-1600END)/1600END input-bit maping/Digital input CH1-bit5
//     PlcTask Inputs/G_IO.arDI[53]/Ch[6] <-> Module 4 (GL20-1600END)/1600END input-bit maping/Digital input CH1-bit6
//     PlcTask Inputs/G_IO.arDI[53]/Ch[7] <-> Module 4 (GL20-1600END)/1600END input-bit maping/Digital input CH1-bit7
//     PlcTask Inputs/G_IO.arDI[53]/Ch[8] <-> Module 4 (GL20-1600END)/1600END input-bit maping/Digital input CH2-bit0
//     PlcTask Inputs/G_IO.arDI[53]/Ch[9] <-> Module 4 (GL20-1600END)/1600END input-bit maping/Digital input CH2-bit1
//     PlcTask Inputs/G_IO.arDI[54]/Ch[0] <-> Module 5 (GL20-1600END)/1600END input-bit maping/Digital input CH1-bit0
//     PlcTask Inputs/G_IO.arDI[54]/Ch[10] <-> Module 5 (GL20-1600END)/1600END input-bit maping/Digital input CH2-bit2
//     PlcTask Inputs/G_IO.arDI[54]/Ch[11] <-> Module 5 (GL20-1600END)/1600END input-bit maping/Digital input CH2-bit3
//     PlcTask Inputs/G_IO.arDI[54]/Ch[12] <-> Module 5 (GL20-1600END)/1600END input-bit maping/Digital input CH2-bit4
//     PlcTask Inputs/G_IO.arDI[54]/Ch[13] <-> Module 5 (GL20-1600END)/1600END input-bit maping/Digital input CH2-bit5
//     PlcTask Inputs/G_IO.arDI[54]/Ch[14] <-> Module 5 (GL20-1600END)/1600END input-bit maping/Digital input CH2-bit6
//     PlcTask Inputs/G_IO.arDI[54]/Ch[15] <-> Module 5 (GL20-1600END)/1600END input-bit maping/Digital input CH2-bit7
//     PlcTask Inputs/G_IO.arDI[54]/Ch[1] <-> Module 5 (GL20-1600END)/1600END input-bit maping/Digital input CH1-bit1
//     PlcTask Inputs/G_IO.arDI[54]/Ch[2] <-> Module 5 (GL20-1600END)/1600END input-bit maping/Digital input CH1-bit2
//     PlcTask Inputs/G_IO.arDI[54]/Ch[3] <-> Module 5 (GL20-1600END)/1600END input-bit maping/Digital input CH1-bit3
//     PlcTask Inputs/G_IO.arDI[54]/Ch[4] <-> Module 5 (GL20-1600END)/1600END input-bit maping/Digital input CH1-bit4
//     PlcTask Inputs/G_IO.arDI[54]/Ch[5] <-> Module 5 (GL20-1600END)/1600END input-bit maping/Digital input CH1-bit5
//     PlcTask Inputs/G_IO.arDI[54]/Ch[6] <-> Module 5 (GL20-1600END)/1600END input-bit maping/Digital input CH1-bit6
//     PlcTask Inputs/G_IO.arDI[54]/Ch[7] <-> Module 5 (GL20-1600END)/1600END input-bit maping/Digital input CH1-bit7
//     PlcTask Inputs/G_IO.arDI[54]/Ch[8] <-> Module 5 (GL20-1600END)/1600END input-bit maping/Digital input CH2-bit0
//     PlcTask Inputs/G_IO.arDI[54]/Ch[9] <-> Module 5 (GL20-1600END)/1600END input-bit maping/Digital input CH2-bit1
//     PlcTask Outputs/G_IO.arDO[50]/Ch[0] <-> Module 6 (GL20-0016ETP)/0016ETP Output-bit maping/Digital output CH1-bit0
//     PlcTask Outputs/G_IO.arDO[50]/Ch[10] <-> Module 6 (GL20-0016ETP)/0016ETP Output-bit maping/Digital output CH2-bit2
//     PlcTask Outputs/G_IO.arDO[50]/Ch[11] <-> Module 6 (GL20-0016ETP)/0016ETP Output-bit maping/Digital output CH2-bit3
//     PlcTask Outputs/G_IO.arDO[50]/Ch[12] <-> Module 6 (GL20-0016ETP)/0016ETP Output-bit maping/Digital output CH2-bit4
//     PlcTask Outputs/G_IO.arDO[50]/Ch[13] <-> Module 6 (GL20-0016ETP)/0016ETP Output-bit maping/Digital output CH2-bit5
//     PlcTask Outputs/G_IO.arDO[50]/Ch[14] <-> Module 6 (GL20-0016ETP)/0016ETP Output-bit maping/Digital output CH2-bit6
//     PlcTask Outputs/G_IO.arDO[50]/Ch[15] <-> Module 6 (GL20-0016ETP)/0016ETP Output-bit maping/Digital output CH2-bit7
//     PlcTask Outputs/G_IO.arDO[50]/Ch[1] <-> Module 6 (GL20-0016ETP)/0016ETP Output-bit maping/Digital output CH1-bit1
//     PlcTask Outputs/G_IO.arDO[50]/Ch[2] <-> Module 6 (GL20-0016ETP)/0016ETP Output-bit maping/Digital output CH1-bit2
//     PlcTask Outputs/G_IO.arDO[50]/Ch[3] <-> Module 6 (GL20-0016ETP)/0016ETP Output-bit maping/Digital output CH1-bit3
//     PlcTask Outputs/G_IO.arDO[50]/Ch[4] <-> Module 6 (GL20-0016ETP)/0016ETP Output-bit maping/Digital output CH1-bit4
//     PlcTask Outputs/G_IO.arDO[50]/Ch[5] <-> Module 6 (GL20-0016ETP)/0016ETP Output-bit maping/Digital output CH1-bit5
//     PlcTask Outputs/G_IO.arDO[50]/Ch[6] <-> Module 6 (GL20-0016ETP)/0016ETP Output-bit maping/Digital output CH1-bit6
//     PlcTask Outputs/G_IO.arDO[50]/Ch[7] <-> Module 6 (GL20-0016ETP)/0016ETP Output-bit maping/Digital output CH1-bit7
//     PlcTask Outputs/G_IO.arDO[50]/Ch[8] <-> Module 6 (GL20-0016ETP)/0016ETP Output-bit maping/Digital output CH2-bit0
//     PlcTask Outputs/G_IO.arDO[50]/Ch[9] <-> Module 6 (GL20-0016ETP)/0016ETP Output-bit maping/Digital output CH2-bit1
//     PlcTask Outputs/G_IO.arDO[51]/Ch[0] <-> Module 7 (GL20-0016ETP)/0016ETP Output-bit maping/Digital output CH1-bit0
//     PlcTask Outputs/G_IO.arDO[51]/Ch[10] <-> Module 7 (GL20-0016ETP)/0016ETP Output-bit maping/Digital output CH2-bit2
//     PlcTask Outputs/G_IO.arDO[51]/Ch[11] <-> Module 7 (GL20-0016ETP)/0016ETP Output-bit maping/Digital output CH2-bit3
//     PlcTask Outputs/G_IO.arDO[51]/Ch[12] <-> Module 7 (GL20-0016ETP)/0016ETP Output-bit maping/Digital output CH2-bit4
//     PlcTask Outputs/G_IO.arDO[51]/Ch[13] <-> Module 7 (GL20-0016ETP)/0016ETP Output-bit maping/Digital output CH2-bit5
//     PlcTask Outputs/G_IO.arDO[51]/Ch[14] <-> Module 7 (GL20-0016ETP)/0016ETP Output-bit maping/Digital output CH2-bit6
//     PlcTask Outputs/G_IO.arDO[51]/Ch[15] <-> Module 7 (GL20-0016ETP)/0016ETP Output-bit maping/Digital output CH2-bit7
//     PlcTask Outputs/G_IO.arDO[51]/Ch[1] <-> Module 7 (GL20-0016ETP)/0016ETP Output-bit maping/Digital output CH1-bit1
//     PlcTask Outputs/G_IO.arDO[51]/Ch[2] <-> Module 7 (GL20-0016ETP)/0016ETP Output-bit maping/Digital output CH1-bit2
//     PlcTask Outputs/G_IO.arDO[51]/Ch[3] <-> Module 7 (GL20-0016ETP)/0016ETP Output-bit maping/Digital output CH1-bit3
//     PlcTask Outputs/G_IO.arDO[51]/Ch[4] <-> Module 7 (GL20-0016ETP)/0016ETP Output-bit maping/Digital output CH1-bit4
//     PlcTask Outputs/G_IO.arDO[51]/Ch[5] <-> Module 7 (GL20-0016ETP)/0016ETP Output-bit maping/Digital output CH1-bit5
//     PlcTask Outputs/G_IO.arDO[51]/Ch[6] <-> Module 7 (GL20-0016ETP)/0016ETP Output-bit maping/Digital output CH1-bit6
//     PlcTask Outputs/G_IO.arDO[51]/Ch[7] <-> Module 7 (GL20-0016ETP)/0016ETP Output-bit maping/Digital output CH1-bit7
//     PlcTask Outputs/G_IO.arDO[51]/Ch[8] <-> Module 7 (GL20-0016ETP)/0016ETP Output-bit maping/Digital output CH2-bit0
//     PlcTask Outputs/G_IO.arDO[51]/Ch[9] <-> Module 7 (GL20-0016ETP)/0016ETP Output-bit maping/Digital output CH2-bit1
//   kittingDeca/kittingDeca Instance <-> pm side/pm0_1_innerConv
//     PlcTask Inputs/GVL.pm[0].inConv.belt[0].fbconverter.running_freq <-> Axis#1 Iutputs/Axis1 Running frequency
//     PlcTask Inputs/GVL.pm[0].inConv.belt[1].fbconverter.running_freq <-> Axis#2 Iutputs/Axis2 Running frequency
//     PlcTask Inputs/GVL.pm[0].inConv.belt[2].fbconverter.running_freq <-> Axis#3 Iutputs/Axis3 Running frequency
//     PlcTask Inputs/GVL.pm[1].inConv.belt[0].fbconverter.running_freq <-> Axis#4 Iutputs/Axis4 Running frequency
//     PlcTask Inputs/GVL.pm[1].inConv.belt[1].fbconverter.running_freq <-> Axis#5 Iutputs/Axis5 Running frequency
//     PlcTask Inputs/GVL.pm[1].inConv.belt[2].fbconverter.running_freq <-> Axis#6 Iutputs/Axis6 Running frequency
//     PlcTask Inputs/GVL.pm[0].inConv.belt[0].fbconverter.status <-> Axis#1 Iutputs/Axis1 AC drive running status word 2
//     PlcTask Inputs/GVL.pm[0].inConv.belt[1].fbconverter.status <-> Axis#2 Iutputs/Axis2 AC drive running status word 2
//     PlcTask Inputs/GVL.pm[0].inConv.belt[2].fbconverter.status <-> Axis#3 Iutputs/Axis3 AC drive running status word 2
//     PlcTask Inputs/GVL.pm[1].inConv.belt[0].fbconverter.status <-> Axis#4 Iutputs/Axis4 AC drive running status word 2
//     PlcTask Inputs/GVL.pm[1].inConv.belt[1].fbconverter.status <-> Axis#5 Iutputs/Axis5 AC drive running status word 2
//     PlcTask Inputs/GVL.pm[1].inConv.belt[2].fbconverter.status <-> Axis#6 Iutputs/Axis6 AC drive running status word 2
//     PlcTask Outputs/GVL.pm[0].inConv.belt[0].fbconverter.cmd <-> Axis#1 Outputs/Axis1 Communication control command
//     PlcTask Outputs/GVL.pm[0].inConv.belt[1].fbconverter.cmd <-> Axis#2 Outputs/Axis2 Communication control command
//     PlcTask Outputs/GVL.pm[0].inConv.belt[2].fbconverter.cmd <-> Axis#3 Outputs/Axis3 Communication control command
//     PlcTask Outputs/GVL.pm[1].inConv.belt[0].fbconverter.cmd <-> Axis#4 Outputs/Axis4 Communication control command
//     PlcTask Outputs/GVL.pm[1].inConv.belt[1].fbconverter.cmd <-> Axis#5 Outputs/Axis5 Communication control command
//     PlcTask Outputs/GVL.pm[1].inConv.belt[2].fbconverter.cmd <-> Axis#6 Outputs/Axis6 Communication control command
//     PlcTask Outputs/GVL.pm[0].inConv.belt[0].fbconverter.freq <-> Axis#1 Outputs/Axis1 Frequency set through communication
//     PlcTask Outputs/GVL.pm[0].inConv.belt[1].fbconverter.freq <-> Axis#2 Outputs/Axis2 Frequency set through communication
//     PlcTask Outputs/GVL.pm[0].inConv.belt[2].fbconverter.freq <-> Axis#3 Outputs/Axis3 Frequency set through communication
//     PlcTask Outputs/GVL.pm[1].inConv.belt[0].fbconverter.freq <-> Axis#4 Outputs/Axis4 Frequency set through communication
//     PlcTask Outputs/GVL.pm[1].inConv.belt[1].fbconverter.freq <-> Axis#5 Outputs/Axis5 Frequency set through communication
//     PlcTask Outputs/GVL.pm[1].inConv.belt[2].fbconverter.freq <-> Axis#6 Outputs/Axis6 Frequency set through communication
//   kittingDeca/kittingDeca Instance <-> pm side/pm0_1_outerConv
//     PlcTask Inputs/GVL.pm[0].outConv.belt[0].fbconverter.running_freq <-> Axis#1 Iutputs/Axis1 Running frequency
//     PlcTask Inputs/GVL.pm[0].outConv.belt[1].fbconverter.running_freq <-> Axis#2 Iutputs/Axis2 Running frequency
//     PlcTask Inputs/GVL.pm[1].outConv.belt[0].fbconverter.running_freq <-> Axis#3 Iutputs/Axis3 Running frequency
//     PlcTask Inputs/GVL.pm[1].outConv.belt[1].fbconverter.running_freq <-> Axis#4 Iutputs/Axis4 Running frequency
//     PlcTask Inputs/GVL.pm[0].outConv.belt[0].fbconverter.status <-> Axis#1 Iutputs/Axis1 AC drive running status word 2
//     PlcTask Inputs/GVL.pm[0].outConv.belt[1].fbconverter.status <-> Axis#2 Iutputs/Axis2 AC drive running status word 2
//     PlcTask Inputs/GVL.pm[1].outConv.belt[0].fbconverter.status <-> Axis#3 Iutputs/Axis3 AC drive running status word 2
//     PlcTask Inputs/GVL.pm[1].outConv.belt[1].fbconverter.status <-> Axis#4 Iutputs/Axis4 AC drive running status word 2
//     PlcTask Outputs/GVL.pm[0].outConv.belt[0].fbconverter.cmd <-> Axis#1 Outputs/Axis1 Communication control command
//     PlcTask Outputs/GVL.pm[0].outConv.belt[1].fbconverter.cmd <-> Axis#2 Outputs/Axis2 Communication control command
//     PlcTask Outputs/GVL.pm[1].outConv.belt[0].fbconverter.cmd <-> Axis#3 Outputs/Axis3 Communication control command
//     PlcTask Outputs/GVL.pm[1].outConv.belt[1].fbconverter.cmd <-> Axis#4 Outputs/Axis4 Communication control command
//     PlcTask Outputs/GVL.pm[0].outConv.belt[0].fbconverter.freq <-> Axis#1 Outputs/Axis1 Frequency set through communication
//     PlcTask Outputs/GVL.pm[0].outConv.belt[1].fbconverter.freq <-> Axis#2 Outputs/Axis2 Frequency set through communication
//     PlcTask Outputs/GVL.pm[1].outConv.belt[0].fbconverter.freq <-> Axis#3 Outputs/Axis3 Frequency set through communication
//     PlcTask Outputs/GVL.pm[1].outConv.belt[1].fbconverter.freq <-> Axis#4 Outputs/Axis4 Frequency set through communication
//   kittingDeca/kittingDeca Instance <-> pm side/pm2_3_dio
//     PlcTask Inputs/G_IO.arDI[55]/Ch[0] <-> Module 1 (GL20-1600END)/1600END input-bit maping/Digital input CH1-bit0
//     PlcTask Inputs/G_IO.arDI[55]/Ch[10] <-> Module 1 (GL20-1600END)/1600END input-bit maping/Digital input CH2-bit2
//     PlcTask Inputs/G_IO.arDI[55]/Ch[11] <-> Module 1 (GL20-1600END)/1600END input-bit maping/Digital input CH2-bit3
//     PlcTask Inputs/G_IO.arDI[55]/Ch[12] <-> Module 1 (GL20-1600END)/1600END input-bit maping/Digital input CH2-bit4
//     PlcTask Inputs/G_IO.arDI[55]/Ch[13] <-> Module 1 (GL20-1600END)/1600END input-bit maping/Digital input CH2-bit5
//     PlcTask Inputs/G_IO.arDI[55]/Ch[14] <-> Module 1 (GL20-1600END)/1600END input-bit maping/Digital input CH2-bit6
//     PlcTask Inputs/G_IO.arDI[55]/Ch[15] <-> Module 1 (GL20-1600END)/1600END input-bit maping/Digital input CH2-bit7
//     PlcTask Inputs/G_IO.arDI[55]/Ch[1] <-> Module 1 (GL20-1600END)/1600END input-bit maping/Digital input CH1-bit1
//     PlcTask Inputs/G_IO.arDI[55]/Ch[2] <-> Module 1 (GL20-1600END)/1600END input-bit maping/Digital input CH1-bit2
//     PlcTask Inputs/G_IO.arDI[55]/Ch[3] <-> Module 1 (GL20-1600END)/1600END input-bit maping/Digital input CH1-bit3
//     PlcTask Inputs/G_IO.arDI[55]/Ch[4] <-> Module 1 (GL20-1600END)/1600END input-bit maping/Digital input CH1-bit4
//     PlcTask Inputs/G_IO.arDI[55]/Ch[5] <-> Module 1 (GL20-1600END)/1600END input-bit maping/Digital input CH1-bit5
//     PlcTask Inputs/G_IO.arDI[55]/Ch[6] <-> Module 1 (GL20-1600END)/1600END input-bit maping/Digital input CH1-bit6
//     PlcTask Inputs/G_IO.arDI[55]/Ch[7] <-> Module 1 (GL20-1600END)/1600END input-bit maping/Digital input CH1-bit7
//     PlcTask Inputs/G_IO.arDI[55]/Ch[8] <-> Module 1 (GL20-1600END)/1600END input-bit maping/Digital input CH2-bit0
//     PlcTask Inputs/G_IO.arDI[55]/Ch[9] <-> Module 1 (GL20-1600END)/1600END input-bit maping/Digital input CH2-bit1
//     PlcTask Inputs/G_IO.arDI[56]/Ch[0] <-> Module 2 (GL20-1600END)/1600END input-bit maping/Digital input CH1-bit0
//     PlcTask Inputs/G_IO.arDI[56]/Ch[10] <-> Module 2 (GL20-1600END)/1600END input-bit maping/Digital input CH2-bit2
//     PlcTask Inputs/G_IO.arDI[56]/Ch[11] <-> Module 2 (GL20-1600END)/1600END input-bit maping/Digital input CH2-bit3
//     PlcTask Inputs/G_IO.arDI[56]/Ch[12] <-> Module 2 (GL20-1600END)/1600END input-bit maping/Digital input CH2-bit4
//     PlcTask Inputs/G_IO.arDI[56]/Ch[13] <-> Module 2 (GL20-1600END)/1600END input-bit maping/Digital input CH2-bit5
//     PlcTask Inputs/G_IO.arDI[56]/Ch[14] <-> Module 2 (GL20-1600END)/1600END input-bit maping/Digital input CH2-bit6
//     PlcTask Inputs/G_IO.arDI[56]/Ch[15] <-> Module 2 (GL20-1600END)/1600END input-bit maping/Digital input CH2-bit7
//     PlcTask Inputs/G_IO.arDI[56]/Ch[1] <-> Module 2 (GL20-1600END)/1600END input-bit maping/Digital input CH1-bit1
//     PlcTask Inputs/G_IO.arDI[56]/Ch[2] <-> Module 2 (GL20-1600END)/1600END input-bit maping/Digital input CH1-bit2
//     PlcTask Inputs/G_IO.arDI[56]/Ch[3] <-> Module 2 (GL20-1600END)/1600END input-bit maping/Digital input CH1-bit3
//     PlcTask Inputs/G_IO.arDI[56]/Ch[4] <-> Module 2 (GL20-1600END)/1600END input-bit maping/Digital input CH1-bit4
//     PlcTask Inputs/G_IO.arDI[56]/Ch[5] <-> Module 2 (GL20-1600END)/1600END input-bit maping/Digital input CH1-bit5
//     PlcTask Inputs/G_IO.arDI[56]/Ch[6] <-> Module 2 (GL20-1600END)/1600END input-bit maping/Digital input CH1-bit6
//     PlcTask Inputs/G_IO.arDI[56]/Ch[7] <-> Module 2 (GL20-1600END)/1600END input-bit maping/Digital input CH1-bit7
//     PlcTask Inputs/G_IO.arDI[56]/Ch[8] <-> Module 2 (GL20-1600END)/1600END input-bit maping/Digital input CH2-bit0
//     PlcTask Inputs/G_IO.arDI[56]/Ch[9] <-> Module 2 (GL20-1600END)/1600END input-bit maping/Digital input CH2-bit1
//     PlcTask Inputs/G_IO.arDI[57]/Ch[0] <-> Module 3 (GL20-1600END)/1600END input-bit maping/Digital input CH1-bit0
//     PlcTask Inputs/G_IO.arDI[57]/Ch[10] <-> Module 3 (GL20-1600END)/1600END input-bit maping/Digital input CH2-bit2
//     PlcTask Inputs/G_IO.arDI[57]/Ch[11] <-> Module 3 (GL20-1600END)/1600END input-bit maping/Digital input CH2-bit3
//     PlcTask Inputs/G_IO.arDI[57]/Ch[12] <-> Module 3 (GL20-1600END)/1600END input-bit maping/Digital input CH2-bit4
//     PlcTask Inputs/G_IO.arDI[57]/Ch[13] <-> Module 3 (GL20-1600END)/1600END input-bit maping/Digital input CH2-bit5
//     PlcTask Inputs/G_IO.arDI[57]/Ch[14] <-> Module 3 (GL20-1600END)/1600END input-bit maping/Digital input CH2-bit6
//     PlcTask Inputs/G_IO.arDI[57]/Ch[15] <-> Module 3 (GL20-1600END)/1600END input-bit maping/Digital input CH2-bit7
//     PlcTask Inputs/G_IO.arDI[57]/Ch[1] <-> Module 3 (GL20-1600END)/1600END input-bit maping/Digital input CH1-bit1
//     PlcTask Inputs/G_IO.arDI[57]/Ch[2] <-> Module 3 (GL20-1600END)/1600END input-bit maping/Digital input CH1-bit2
//     PlcTask Inputs/G_IO.arDI[57]/Ch[3] <-> Module 3 (GL20-1600END)/1600END input-bit maping/Digital input CH1-bit3
//     PlcTask Inputs/G_IO.arDI[57]/Ch[4] <-> Module 3 (GL20-1600END)/1600END input-bit maping/Digital input CH1-bit4
//     PlcTask Inputs/G_IO.arDI[57]/Ch[5] <-> Module 3 (GL20-1600END)/1600END input-bit maping/Digital input CH1-bit5
//     PlcTask Inputs/G_IO.arDI[57]/Ch[6] <-> Module 3 (GL20-1600END)/1600END input-bit maping/Digital input CH1-bit6
//     PlcTask Inputs/G_IO.arDI[57]/Ch[7] <-> Module 3 (GL20-1600END)/1600END input-bit maping/Digital input CH1-bit7
//     PlcTask Inputs/G_IO.arDI[57]/Ch[8] <-> Module 3 (GL20-1600END)/1600END input-bit maping/Digital input CH2-bit0
//     PlcTask Inputs/G_IO.arDI[57]/Ch[9] <-> Module 3 (GL20-1600END)/1600END input-bit maping/Digital input CH2-bit1
//     PlcTask Inputs/G_IO.arDI[58]/Ch[0] <-> Module 4 (GL20-1600END)/1600END input-bit maping/Digital input CH1-bit0
//     PlcTask Inputs/G_IO.arDI[58]/Ch[10] <-> Module 4 (GL20-1600END)/1600END input-bit maping/Digital input CH2-bit2
//     PlcTask Inputs/G_IO.arDI[58]/Ch[11] <-> Module 4 (GL20-1600END)/1600END input-bit maping/Digital input CH2-bit3
//     PlcTask Inputs/G_IO.arDI[58]/Ch[12] <-> Module 4 (GL20-1600END)/1600END input-bit maping/Digital input CH2-bit4
//     PlcTask Inputs/G_IO.arDI[58]/Ch[13] <-> Module 4 (GL20-1600END)/1600END input-bit maping/Digital input CH2-bit5
//     PlcTask Inputs/G_IO.arDI[58]/Ch[14] <-> Module 4 (GL20-1600END)/1600END input-bit maping/Digital input CH2-bit6
//     PlcTask Inputs/G_IO.arDI[58]/Ch[15] <-> Module 4 (GL20-1600END)/1600END input-bit maping/Digital input CH2-bit7
//     PlcTask Inputs/G_IO.arDI[58]/Ch[1] <-> Module 4 (GL20-1600END)/1600END input-bit maping/Digital input CH1-bit1
//     PlcTask Inputs/G_IO.arDI[58]/Ch[2] <-> Module 4 (GL20-1600END)/1600END input-bit maping/Digital input CH1-bit2
//     PlcTask Inputs/G_IO.arDI[58]/Ch[3] <-> Module 4 (GL20-1600END)/1600END input-bit maping/Digital input CH1-bit3
//     PlcTask Inputs/G_IO.arDI[58]/Ch[4] <-> Module 4 (GL20-1600END)/1600END input-bit maping/Digital input CH1-bit4
//     PlcTask Inputs/G_IO.arDI[58]/Ch[5] <-> Module 4 (GL20-1600END)/1600END input-bit maping/Digital input CH1-bit5
//     PlcTask Inputs/G_IO.arDI[58]/Ch[6] <-> Module 4 (GL20-1600END)/1600END input-bit maping/Digital input CH1-bit6
//     PlcTask Inputs/G_IO.arDI[58]/Ch[7] <-> Module 4 (GL20-1600END)/1600END input-bit maping/Digital input CH1-bit7
//     PlcTask Inputs/G_IO.arDI[58]/Ch[8] <-> Module 4 (GL20-1600END)/1600END input-bit maping/Digital input CH2-bit0
//     PlcTask Inputs/G_IO.arDI[58]/Ch[9] <-> Module 4 (GL20-1600END)/1600END input-bit maping/Digital input CH2-bit1
//     PlcTask Inputs/G_IO.arDI[59]/Ch[0] <-> Module 5 (GL20-1600END)/1600END input-bit maping/Digital input CH1-bit0
//     PlcTask Inputs/G_IO.arDI[59]/Ch[10] <-> Module 5 (GL20-1600END)/1600END input-bit maping/Digital input CH2-bit2
//     PlcTask Inputs/G_IO.arDI[59]/Ch[11] <-> Module 5 (GL20-1600END)/1600END input-bit maping/Digital input CH2-bit3
//     PlcTask Inputs/G_IO.arDI[59]/Ch[12] <-> Module 5 (GL20-1600END)/1600END input-bit maping/Digital input CH2-bit4
//     PlcTask Inputs/G_IO.arDI[59]/Ch[13] <-> Module 5 (GL20-1600END)/1600END input-bit maping/Digital input CH2-bit5
//     PlcTask Inputs/G_IO.arDI[59]/Ch[14] <-> Module 5 (GL20-1600END)/1600END input-bit maping/Digital input CH2-bit6
//     PlcTask Inputs/G_IO.arDI[59]/Ch[15] <-> Module 5 (GL20-1600END)/1600END input-bit maping/Digital input CH2-bit7
//     PlcTask Inputs/G_IO.arDI[59]/Ch[1] <-> Module 5 (GL20-1600END)/1600END input-bit maping/Digital input CH1-bit1
//     PlcTask Inputs/G_IO.arDI[59]/Ch[2] <-> Module 5 (GL20-1600END)/1600END input-bit maping/Digital input CH1-bit2
//     PlcTask Inputs/G_IO.arDI[59]/Ch[3] <-> Module 5 (GL20-1600END)/1600END input-bit maping/Digital input CH1-bit3
//     PlcTask Inputs/G_IO.arDI[59]/Ch[4] <-> Module 5 (GL20-1600END)/1600END input-bit maping/Digital input CH1-bit4
//     PlcTask Inputs/G_IO.arDI[59]/Ch[5] <-> Module 5 (GL20-1600END)/1600END input-bit maping/Digital input CH1-bit5
//     PlcTask Inputs/G_IO.arDI[59]/Ch[6] <-> Module 5 (GL20-1600END)/1600END input-bit maping/Digital input CH1-bit6
//     PlcTask Inputs/G_IO.arDI[59]/Ch[7] <-> Module 5 (GL20-1600END)/1600END input-bit maping/Digital input CH1-bit7
//     PlcTask Inputs/G_IO.arDI[59]/Ch[8] <-> Module 5 (GL20-1600END)/1600END input-bit maping/Digital input CH2-bit0
//     PlcTask Inputs/G_IO.arDI[59]/Ch[9] <-> Module 5 (GL20-1600END)/1600END input-bit maping/Digital input CH2-bit1
//     PlcTask Inputs/G_IO.arDI[77]/Ch[0] <-> Module 6 (GL20-1600END)/1600END input-bit maping/Digital input CH1-bit0
//     PlcTask Inputs/G_IO.arDI[77]/Ch[10] <-> Module 6 (GL20-1600END)/1600END input-bit maping/Digital input CH2-bit2
//     PlcTask Inputs/G_IO.arDI[77]/Ch[11] <-> Module 6 (GL20-1600END)/1600END input-bit maping/Digital input CH2-bit3
//     PlcTask Inputs/G_IO.arDI[77]/Ch[12] <-> Module 6 (GL20-1600END)/1600END input-bit maping/Digital input CH2-bit4
//     PlcTask Inputs/G_IO.arDI[77]/Ch[13] <-> Module 6 (GL20-1600END)/1600END input-bit maping/Digital input CH2-bit5
//     PlcTask Inputs/G_IO.arDI[77]/Ch[14] <-> Module 6 (GL20-1600END)/1600END input-bit maping/Digital input CH2-bit6
//     PlcTask Inputs/G_IO.arDI[77]/Ch[15] <-> Module 6 (GL20-1600END)/1600END input-bit maping/Digital input CH2-bit7
//     PlcTask Inputs/G_IO.arDI[77]/Ch[1] <-> Module 6 (GL20-1600END)/1600END input-bit maping/Digital input CH1-bit1
//     PlcTask Inputs/G_IO.arDI[77]/Ch[2] <-> Module 6 (GL20-1600END)/1600END input-bit maping/Digital input CH1-bit2
//     PlcTask Inputs/G_IO.arDI[77]/Ch[3] <-> Module 6 (GL20-1600END)/1600END input-bit maping/Digital input CH1-bit3
//     PlcTask Inputs/G_IO.arDI[77]/Ch[4] <-> Module 6 (GL20-1600END)/1600END input-bit maping/Digital input CH1-bit4
//     PlcTask Inputs/G_IO.arDI[77]/Ch[5] <-> Module 6 (GL20-1600END)/1600END input-bit maping/Digital input CH1-bit5
//     PlcTask Inputs/G_IO.arDI[77]/Ch[6] <-> Module 6 (GL20-1600END)/1600END input-bit maping/Digital input CH1-bit6
//     PlcTask Inputs/G_IO.arDI[77]/Ch[7] <-> Module 6 (GL20-1600END)/1600END input-bit maping/Digital input CH1-bit7
//     PlcTask Inputs/G_IO.arDI[77]/Ch[8] <-> Module 6 (GL20-1600END)/1600END input-bit maping/Digital input CH2-bit0
//     PlcTask Inputs/G_IO.arDI[77]/Ch[9] <-> Module 6 (GL20-1600END)/1600END input-bit maping/Digital input CH2-bit1
//     PlcTask Outputs/G_IO.arDO[54]/Ch[0] <-> Module 7 (GL20-0016ETP)/0016ETP Output-bit maping/Digital output CH1-bit0
//     PlcTask Outputs/G_IO.arDO[54]/Ch[10] <-> Module 7 (GL20-0016ETP)/0016ETP Output-bit maping/Digital output CH2-bit2
//     PlcTask Outputs/G_IO.arDO[54]/Ch[11] <-> Module 7 (GL20-0016ETP)/0016ETP Output-bit maping/Digital output CH2-bit3
//     PlcTask Outputs/G_IO.arDO[54]/Ch[12] <-> Module 7 (GL20-0016ETP)/0016ETP Output-bit maping/Digital output CH2-bit4
//     PlcTask Outputs/G_IO.arDO[54]/Ch[13] <-> Module 7 (GL20-0016ETP)/0016ETP Output-bit maping/Digital output CH2-bit5
//     PlcTask Outputs/G_IO.arDO[54]/Ch[14] <-> Module 7 (GL20-0016ETP)/0016ETP Output-bit maping/Digital output CH2-bit6
//     PlcTask Outputs/G_IO.arDO[54]/Ch[15] <-> Module 7 (GL20-0016ETP)/0016ETP Output-bit maping/Digital output CH2-bit7
//     PlcTask Outputs/G_IO.arDO[54]/Ch[1] <-> Module 7 (GL20-0016ETP)/0016ETP Output-bit maping/Digital output CH1-bit1
//     PlcTask Outputs/G_IO.arDO[54]/Ch[2] <-> Module 7 (GL20-0016ETP)/0016ETP Output-bit maping/Digital output CH1-bit2
//     PlcTask Outputs/G_IO.arDO[54]/Ch[3] <-> Module 7 (GL20-0016ETP)/0016ETP Output-bit maping/Digital output CH1-bit3
//     PlcTask Outputs/G_IO.arDO[54]/Ch[4] <-> Module 7 (GL20-0016ETP)/0016ETP Output-bit maping/Digital output CH1-bit4
//     PlcTask Outputs/G_IO.arDO[54]/Ch[5] <-> Module 7 (GL20-0016ETP)/0016ETP Output-bit maping/Digital output CH1-bit5
//     PlcTask Outputs/G_IO.arDO[54]/Ch[6] <-> Module 7 (GL20-0016ETP)/0016ETP Output-bit maping/Digital output CH1-bit6
//     PlcTask Outputs/G_IO.arDO[54]/Ch[7] <-> Module 7 (GL20-0016ETP)/0016ETP Output-bit maping/Digital output CH1-bit7
//     PlcTask Outputs/G_IO.arDO[54]/Ch[8] <-> Module 7 (GL20-0016ETP)/0016ETP Output-bit maping/Digital output CH2-bit0
//     PlcTask Outputs/G_IO.arDO[54]/Ch[9] <-> Module 7 (GL20-0016ETP)/0016ETP Output-bit maping/Digital output CH2-bit1
//     PlcTask Outputs/G_IO.arDO[55]/Ch[0] <-> Module 8 (GL20-0016ETP)/0016ETP Output-bit maping/Digital output CH1-bit0
//     PlcTask Outputs/G_IO.arDO[55]/Ch[10] <-> Module 8 (GL20-0016ETP)/0016ETP Output-bit maping/Digital output CH2-bit2
//     PlcTask Outputs/G_IO.arDO[55]/Ch[11] <-> Module 8 (GL20-0016ETP)/0016ETP Output-bit maping/Digital output CH2-bit3
//     PlcTask Outputs/G_IO.arDO[55]/Ch[12] <-> Module 8 (GL20-0016ETP)/0016ETP Output-bit maping/Digital output CH2-bit4
//     PlcTask Outputs/G_IO.arDO[55]/Ch[13] <-> Module 8 (GL20-0016ETP)/0016ETP Output-bit maping/Digital output CH2-bit5
//     PlcTask Outputs/G_IO.arDO[55]/Ch[14] <-> Module 8 (GL20-0016ETP)/0016ETP Output-bit maping/Digital output CH2-bit6
//     PlcTask Outputs/G_IO.arDO[55]/Ch[15] <-> Module 8 (GL20-0016ETP)/0016ETP Output-bit maping/Digital output CH2-bit7
//     PlcTask Outputs/G_IO.arDO[55]/Ch[1] <-> Module 8 (GL20-0016ETP)/0016ETP Output-bit maping/Digital output CH1-bit1
//     PlcTask Outputs/G_IO.arDO[55]/Ch[2] <-> Module 8 (GL20-0016ETP)/0016ETP Output-bit maping/Digital output CH1-bit2
//     PlcTask Outputs/G_IO.arDO[55]/Ch[3] <-> Module 8 (GL20-0016ETP)/0016ETP Output-bit maping/Digital output CH1-bit3
//     PlcTask Outputs/G_IO.arDO[55]/Ch[4] <-> Module 8 (GL20-0016ETP)/0016ETP Output-bit maping/Digital output CH1-bit4
//     PlcTask Outputs/G_IO.arDO[55]/Ch[5] <-> Module 8 (GL20-0016ETP)/0016ETP Output-bit maping/Digital output CH1-bit5
//     PlcTask Outputs/G_IO.arDO[55]/Ch[6] <-> Module 8 (GL20-0016ETP)/0016ETP Output-bit maping/Digital output CH1-bit6
//     PlcTask Outputs/G_IO.arDO[55]/Ch[7] <-> Module 8 (GL20-0016ETP)/0016ETP Output-bit maping/Digital output CH1-bit7
//     PlcTask Outputs/G_IO.arDO[55]/Ch[8] <-> Module 8 (GL20-0016ETP)/0016ETP Output-bit maping/Digital output CH2-bit0
//     PlcTask Outputs/G_IO.arDO[55]/Ch[9] <-> Module 8 (GL20-0016ETP)/0016ETP Output-bit maping/Digital output CH2-bit1
//   kittingDeca/kittingDeca Instance <-> pm side/pm2_3_innerConv
//     PlcTask Inputs/GVL.pm[2].inConv.belt[0].fbconverter.running_freq <-> Axis#1 Iutputs/Axis1 Running frequency
//     PlcTask Inputs/GVL.pm[2].inConv.belt[1].fbconverter.running_freq <-> Axis#2 Iutputs/Axis2 Running frequency
//     PlcTask Inputs/GVL.pm[2].inConv.belt[2].fbconverter.running_freq <-> Axis#3 Iutputs/Axis3 Running frequency
//     PlcTask Inputs/GVL.pm[3].inConv.belt[0].fbconverter.running_freq <-> Axis#4 Iutputs/Axis4 Running frequency
//     PlcTask Inputs/GVL.pm[3].inConv.belt[1].fbconverter.running_freq <-> Axis#5 Iutputs/Axis5 Running frequency
//     PlcTask Inputs/GVL.pm[3].inConv.belt[2].fbconverter.running_freq <-> Axis#6 Iutputs/Axis6 Running frequency
//     PlcTask Inputs/GVL.pm[2].inConv.belt[0].fbconverter.status <-> Axis#1 Iutputs/Axis1 AC drive running status word 2
//     PlcTask Inputs/GVL.pm[2].inConv.belt[1].fbconverter.status <-> Axis#2 Iutputs/Axis2 AC drive running status word 2
//     PlcTask Inputs/GVL.pm[2].inConv.belt[2].fbconverter.status <-> Axis#3 Iutputs/Axis3 AC drive running status word 2
//     PlcTask Inputs/GVL.pm[3].inConv.belt[0].fbconverter.status <-> Axis#4 Iutputs/Axis4 AC drive running status word 2
//     PlcTask Inputs/GVL.pm[3].inConv.belt[1].fbconverter.status <-> Axis#5 Iutputs/Axis5 AC drive running status word 2
//     PlcTask Inputs/GVL.pm[3].inConv.belt[2].fbconverter.status <-> Axis#6 Iutputs/Axis6 AC drive running status word 2
//     PlcTask Outputs/GVL.pm[2].inConv.belt[0].fbconverter.cmd <-> Axis#1 Outputs/Axis1 Communication control command
//     PlcTask Outputs/GVL.pm[2].inConv.belt[1].fbconverter.cmd <-> Axis#2 Outputs/Axis2 Communication control command
//     PlcTask Outputs/GVL.pm[2].inConv.belt[2].fbconverter.cmd <-> Axis#3 Outputs/Axis3 Communication control command
//     PlcTask Outputs/GVL.pm[3].inConv.belt[0].fbconverter.cmd <-> Axis#4 Outputs/Axis4 Communication control command
//     PlcTask Outputs/GVL.pm[3].inConv.belt[1].fbconverter.cmd <-> Axis#5 Outputs/Axis5 Communication control command
//     PlcTask Outputs/GVL.pm[3].inConv.belt[2].fbconverter.cmd <-> Axis#6 Outputs/Axis6 Communication control command
//     PlcTask Outputs/GVL.pm[2].inConv.belt[0].fbconverter.freq <-> Axis#1 Outputs/Axis1 Frequency set through communication
//     PlcTask Outputs/GVL.pm[2].inConv.belt[1].fbconverter.freq <-> Axis#2 Outputs/Axis2 Frequency set through communication
//     PlcTask Outputs/GVL.pm[2].inConv.belt[2].fbconverter.freq <-> Axis#3 Outputs/Axis3 Frequency set through communication
//     PlcTask Outputs/GVL.pm[3].inConv.belt[0].fbconverter.freq <-> Axis#4 Outputs/Axis4 Frequency set through communication
//     PlcTask Outputs/GVL.pm[3].inConv.belt[1].fbconverter.freq <-> Axis#5 Outputs/Axis5 Frequency set through communication
//     PlcTask Outputs/GVL.pm[3].inConv.belt[2].fbconverter.freq <-> Axis#6 Outputs/Axis6 Frequency set through communication
//   kittingDeca/kittingDeca Instance <-> pm side/pm2_3_outerConv
//     PlcTask Inputs/GVL.pm[2].outConv.belt[0].fbconverter.running_freq <-> Axis#1 Iutputs/Axis1 Running frequency
//     PlcTask Inputs/GVL.pm[2].outConv.belt[1].fbconverter.running_freq <-> Axis#2 Iutputs/Axis2 Running frequency
//     PlcTask Inputs/GVL.pm[3].outConv.belt[0].fbconverter.running_freq <-> Axis#3 Iutputs/Axis3 Running frequency
//     PlcTask Inputs/GVL.pm[3].outConv.belt[1].fbconverter.running_freq <-> Axis#4 Iutputs/Axis4 Running frequency
//     PlcTask Inputs/GVL.pm[2].outConv.belt[0].fbconverter.status <-> Axis#1 Iutputs/Axis1 AC drive running status word 2
//     PlcTask Inputs/GVL.pm[2].outConv.belt[1].fbconverter.status <-> Axis#2 Iutputs/Axis2 AC drive running status word 2
//     PlcTask Inputs/GVL.pm[3].outConv.belt[0].fbconverter.status <-> Axis#3 Iutputs/Axis3 AC drive running status word 2
//     PlcTask Inputs/GVL.pm[3].outConv.belt[1].fbconverter.status <-> Axis#4 Iutputs/Axis4 AC drive running status word 2
//     PlcTask Outputs/GVL.pm[2].outConv.belt[0].fbconverter.cmd <-> Axis#1 Outputs/Axis1 Communication control command
//     PlcTask Outputs/GVL.pm[2].outConv.belt[1].fbconverter.cmd <-> Axis#2 Outputs/Axis2 Communication control command
//     PlcTask Outputs/GVL.pm[3].outConv.belt[0].fbconverter.cmd <-> Axis#3 Outputs/Axis3 Communication control command
//     PlcTask Outputs/GVL.pm[3].outConv.belt[1].fbconverter.cmd <-> Axis#4 Outputs/Axis4 Communication control command
//     PlcTask Outputs/GVL.pm[2].outConv.belt[0].fbconverter.freq <-> Axis#1 Outputs/Axis1 Frequency set through communication
//     PlcTask Outputs/GVL.pm[2].outConv.belt[1].fbconverter.freq <-> Axis#2 Outputs/Axis2 Frequency set through communication
//     PlcTask Outputs/GVL.pm[3].outConv.belt[0].fbconverter.freq <-> Axis#3 Outputs/Axis3 Frequency set through communication
//     PlcTask Outputs/GVL.pm[3].outConv.belt[1].fbconverter.freq <-> Axis#4 Outputs/Axis4 Frequency set through communication
//   kittingDeca/kittingDeca Instance <-> pm side/pm4_5_dio
//     PlcTask Inputs/G_IO.arDI[60]/Ch[0] <-> Module 1 (GL20-1600END)/1600END input-bit maping/Digital input CH1-bit0
//     PlcTask Inputs/G_IO.arDI[60]/Ch[10] <-> Module 1 (GL20-1600END)/1600END input-bit maping/Digital input CH2-bit2
//     PlcTask Inputs/G_IO.arDI[60]/Ch[11] <-> Module 1 (GL20-1600END)/1600END input-bit maping/Digital input CH2-bit3
//     PlcTask Inputs/G_IO.arDI[60]/Ch[12] <-> Module 1 (GL20-1600END)/1600END input-bit maping/Digital input CH2-bit4
//     PlcTask Inputs/G_IO.arDI[60]/Ch[13] <-> Module 1 (GL20-1600END)/1600END input-bit maping/Digital input CH2-bit5
//     PlcTask Inputs/G_IO.arDI[60]/Ch[14] <-> Module 1 (GL20-1600END)/1600END input-bit maping/Digital input CH2-bit6
//     PlcTask Inputs/G_IO.arDI[60]/Ch[15] <-> Module 1 (GL20-1600END)/1600END input-bit maping/Digital input CH2-bit7
//     PlcTask Inputs/G_IO.arDI[60]/Ch[1] <-> Module 1 (GL20-1600END)/1600END input-bit maping/Digital input CH1-bit1
//     PlcTask Inputs/G_IO.arDI[60]/Ch[2] <-> Module 1 (GL20-1600END)/1600END input-bit maping/Digital input CH1-bit2
//     PlcTask Inputs/G_IO.arDI[60]/Ch[3] <-> Module 1 (GL20-1600END)/1600END input-bit maping/Digital input CH1-bit3
//     PlcTask Inputs/G_IO.arDI[60]/Ch[4] <-> Module 1 (GL20-1600END)/1600END input-bit maping/Digital input CH1-bit4
//     PlcTask Inputs/G_IO.arDI[60]/Ch[5] <-> Module 1 (GL20-1600END)/1600END input-bit maping/Digital input CH1-bit5
//     PlcTask Inputs/G_IO.arDI[60]/Ch[6] <-> Module 1 (GL20-1600END)/1600END input-bit maping/Digital input CH1-bit6
//     PlcTask Inputs/G_IO.arDI[60]/Ch[7] <-> Module 1 (GL20-1600END)/1600END input-bit maping/Digital input CH1-bit7
//     PlcTask Inputs/G_IO.arDI[60]/Ch[8] <-> Module 1 (GL20-1600END)/1600END input-bit maping/Digital input CH2-bit0
//     PlcTask Inputs/G_IO.arDI[60]/Ch[9] <-> Module 1 (GL20-1600END)/1600END input-bit maping/Digital input CH2-bit1
//     PlcTask Inputs/G_IO.arDI[61]/Ch[0] <-> Module 2 (GL20-1600END)/1600END input-bit maping/Digital input CH1-bit0
//     PlcTask Inputs/G_IO.arDI[61]/Ch[10] <-> Module 2 (GL20-1600END)/1600END input-bit maping/Digital input CH2-bit2
//     PlcTask Inputs/G_IO.arDI[61]/Ch[11] <-> Module 2 (GL20-1600END)/1600END input-bit maping/Digital input CH2-bit3
//     PlcTask Inputs/G_IO.arDI[61]/Ch[12] <-> Module 2 (GL20-1600END)/1600END input-bit maping/Digital input CH2-bit4
//     PlcTask Inputs/G_IO.arDI[61]/Ch[13] <-> Module 2 (GL20-1600END)/1600END input-bit maping/Digital input CH2-bit5
//     PlcTask Inputs/G_IO.arDI[61]/Ch[14] <-> Module 2 (GL20-1600END)/1600END input-bit maping/Digital input CH2-bit6
//     PlcTask Inputs/G_IO.arDI[61]/Ch[15] <-> Module 2 (GL20-1600END)/1600END input-bit maping/Digital input CH2-bit7
//     PlcTask Inputs/G_IO.arDI[61]/Ch[1] <-> Module 2 (GL20-1600END)/1600END input-bit maping/Digital input CH1-bit1
//     PlcTask Inputs/G_IO.arDI[61]/Ch[2] <-> Module 2 (GL20-1600END)/1600END input-bit maping/Digital input CH1-bit2
//     PlcTask Inputs/G_IO.arDI[61]/Ch[3] <-> Module 2 (GL20-1600END)/1600END input-bit maping/Digital input CH1-bit3
//     PlcTask Inputs/G_IO.arDI[61]/Ch[4] <-> Module 2 (GL20-1600END)/1600END input-bit maping/Digital input CH1-bit4
//     PlcTask Inputs/G_IO.arDI[61]/Ch[5] <-> Module 2 (GL20-1600END)/1600END input-bit maping/Digital input CH1-bit5
//     PlcTask Inputs/G_IO.arDI[61]/Ch[6] <-> Module 2 (GL20-1600END)/1600END input-bit maping/Digital input CH1-bit6
//     PlcTask Inputs/G_IO.arDI[61]/Ch[7] <-> Module 2 (GL20-1600END)/1600END input-bit maping/Digital input CH1-bit7
//     PlcTask Inputs/G_IO.arDI[61]/Ch[8] <-> Module 2 (GL20-1600END)/1600END input-bit maping/Digital input CH2-bit0
//     PlcTask Inputs/G_IO.arDI[61]/Ch[9] <-> Module 2 (GL20-1600END)/1600END input-bit maping/Digital input CH2-bit1
//     PlcTask Inputs/G_IO.arDI[62]/Ch[0] <-> Module 3 (GL20-1600END)/1600END input-bit maping/Digital input CH1-bit0
//     PlcTask Inputs/G_IO.arDI[62]/Ch[10] <-> Module 3 (GL20-1600END)/1600END input-bit maping/Digital input CH2-bit2
//     PlcTask Inputs/G_IO.arDI[62]/Ch[11] <-> Module 3 (GL20-1600END)/1600END input-bit maping/Digital input CH2-bit3
//     PlcTask Inputs/G_IO.arDI[62]/Ch[12] <-> Module 3 (GL20-1600END)/1600END input-bit maping/Digital input CH2-bit4
//     PlcTask Inputs/G_IO.arDI[62]/Ch[13] <-> Module 3 (GL20-1600END)/1600END input-bit maping/Digital input CH2-bit5
//     PlcTask Inputs/G_IO.arDI[62]/Ch[14] <-> Module 3 (GL20-1600END)/1600END input-bit maping/Digital input CH2-bit6
//     PlcTask Inputs/G_IO.arDI[62]/Ch[15] <-> Module 3 (GL20-1600END)/1600END input-bit maping/Digital input CH2-bit7
//     PlcTask Inputs/G_IO.arDI[62]/Ch[1] <-> Module 3 (GL20-1600END)/1600END input-bit maping/Digital input CH1-bit1
//     PlcTask Inputs/G_IO.arDI[62]/Ch[2] <-> Module 3 (GL20-1600END)/1600END input-bit maping/Digital input CH1-bit2
//     PlcTask Inputs/G_IO.arDI[62]/Ch[3] <-> Module 3 (GL20-1600END)/1600END input-bit maping/Digital input CH1-bit3
//     PlcTask Inputs/G_IO.arDI[62]/Ch[4] <-> Module 3 (GL20-1600END)/1600END input-bit maping/Digital input CH1-bit4
//     PlcTask Inputs/G_IO.arDI[62]/Ch[5] <-> Module 3 (GL20-1600END)/1600END input-bit maping/Digital input CH1-bit5
//     PlcTask Inputs/G_IO.arDI[62]/Ch[6] <-> Module 3 (GL20-1600END)/1600END input-bit maping/Digital input CH1-bit6
//     PlcTask Inputs/G_IO.arDI[62]/Ch[7] <-> Module 3 (GL20-1600END)/1600END input-bit maping/Digital input CH1-bit7
//     PlcTask Inputs/G_IO.arDI[62]/Ch[8] <-> Module 3 (GL20-1600END)/1600END input-bit maping/Digital input CH2-bit0
//     PlcTask Inputs/G_IO.arDI[62]/Ch[9] <-> Module 3 (GL20-1600END)/1600END input-bit maping/Digital input CH2-bit1
//     PlcTask Inputs/G_IO.arDI[63]/Ch[0] <-> Module 4 (GL20-1600END)/1600END input-bit maping/Digital input CH1-bit0
//     PlcTask Inputs/G_IO.arDI[63]/Ch[10] <-> Module 4 (GL20-1600END)/1600END input-bit maping/Digital input CH2-bit2
//     PlcTask Inputs/G_IO.arDI[63]/Ch[11] <-> Module 4 (GL20-1600END)/1600END input-bit maping/Digital input CH2-bit3
//     PlcTask Inputs/G_IO.arDI[63]/Ch[12] <-> Module 4 (GL20-1600END)/1600END input-bit maping/Digital input CH2-bit4
//     PlcTask Inputs/G_IO.arDI[63]/Ch[13] <-> Module 4 (GL20-1600END)/1600END input-bit maping/Digital input CH2-bit5
//     PlcTask Inputs/G_IO.arDI[63]/Ch[14] <-> Module 4 (GL20-1600END)/1600END input-bit maping/Digital input CH2-bit6
//     PlcTask Inputs/G_IO.arDI[63]/Ch[15] <-> Module 4 (GL20-1600END)/1600END input-bit maping/Digital input CH2-bit7
//     PlcTask Inputs/G_IO.arDI[63]/Ch[1] <-> Module 4 (GL20-1600END)/1600END input-bit maping/Digital input CH1-bit1
//     PlcTask Inputs/G_IO.arDI[63]/Ch[2] <-> Module 4 (GL20-1600END)/1600END input-bit maping/Digital input CH1-bit2
//     PlcTask Inputs/G_IO.arDI[63]/Ch[3] <-> Module 4 (GL20-1600END)/1600END input-bit maping/Digital input CH1-bit3
//     PlcTask Inputs/G_IO.arDI[63]/Ch[4] <-> Module 4 (GL20-1600END)/1600END input-bit maping/Digital input CH1-bit4
//     PlcTask Inputs/G_IO.arDI[63]/Ch[5] <-> Module 4 (GL20-1600END)/1600END input-bit maping/Digital input CH1-bit5
//     PlcTask Inputs/G_IO.arDI[63]/Ch[6] <-> Module 4 (GL20-1600END)/1600END input-bit maping/Digital input CH1-bit6
//     PlcTask Inputs/G_IO.arDI[63]/Ch[7] <-> Module 4 (GL20-1600END)/1600END input-bit maping/Digital input CH1-bit7
//     PlcTask Inputs/G_IO.arDI[63]/Ch[8] <-> Module 4 (GL20-1600END)/1600END input-bit maping/Digital input CH2-bit0
//     PlcTask Inputs/G_IO.arDI[63]/Ch[9] <-> Module 4 (GL20-1600END)/1600END input-bit maping/Digital input CH2-bit1
//     PlcTask Inputs/G_IO.arDI[64]/Ch[0] <-> Module 5 (GL20-1600END)/1600END input-bit maping/Digital input CH1-bit0
//     PlcTask Inputs/G_IO.arDI[64]/Ch[10] <-> Module 5 (GL20-1600END)/1600END input-bit maping/Digital input CH2-bit2
//     PlcTask Inputs/G_IO.arDI[64]/Ch[11] <-> Module 5 (GL20-1600END)/1600END input-bit maping/Digital input CH2-bit3
//     PlcTask Inputs/G_IO.arDI[64]/Ch[12] <-> Module 5 (GL20-1600END)/1600END input-bit maping/Digital input CH2-bit4
//     PlcTask Inputs/G_IO.arDI[64]/Ch[13] <-> Module 5 (GL20-1600END)/1600END input-bit maping/Digital input CH2-bit5
//     PlcTask Inputs/G_IO.arDI[64]/Ch[14] <-> Module 5 (GL20-1600END)/1600END input-bit maping/Digital input CH2-bit6
//     PlcTask Inputs/G_IO.arDI[64]/Ch[15] <-> Module 5 (GL20-1600END)/1600END input-bit maping/Digital input CH2-bit7
//     PlcTask Inputs/G_IO.arDI[64]/Ch[1] <-> Module 5 (GL20-1600END)/1600END input-bit maping/Digital input CH1-bit1
//     PlcTask Inputs/G_IO.arDI[64]/Ch[2] <-> Module 5 (GL20-1600END)/1600END input-bit maping/Digital input CH1-bit2
//     PlcTask Inputs/G_IO.arDI[64]/Ch[3] <-> Module 5 (GL20-1600END)/1600END input-bit maping/Digital input CH1-bit3
//     PlcTask Inputs/G_IO.arDI[64]/Ch[4] <-> Module 5 (GL20-1600END)/1600END input-bit maping/Digital input CH1-bit4
//     PlcTask Inputs/G_IO.arDI[64]/Ch[5] <-> Module 5 (GL20-1600END)/1600END input-bit maping/Digital input CH1-bit5
//     PlcTask Inputs/G_IO.arDI[64]/Ch[6] <-> Module 5 (GL20-1600END)/1600END input-bit maping/Digital input CH1-bit6
//     PlcTask Inputs/G_IO.arDI[64]/Ch[7] <-> Module 5 (GL20-1600END)/1600END input-bit maping/Digital input CH1-bit7
//     PlcTask Inputs/G_IO.arDI[64]/Ch[8] <-> Module 5 (GL20-1600END)/1600END input-bit maping/Digital input CH2-bit0
//     PlcTask Inputs/G_IO.arDI[64]/Ch[9] <-> Module 5 (GL20-1600END)/1600END input-bit maping/Digital input CH2-bit1
//     PlcTask Inputs/G_IO.arDI[78]/Ch[0] <-> Module 6 (GL20-1600END)/1600END input-bit maping/Digital input CH1-bit0
//     PlcTask Inputs/G_IO.arDI[78]/Ch[10] <-> Module 6 (GL20-1600END)/1600END input-bit maping/Digital input CH2-bit2
//     PlcTask Inputs/G_IO.arDI[78]/Ch[11] <-> Module 6 (GL20-1600END)/1600END input-bit maping/Digital input CH2-bit3
//     PlcTask Inputs/G_IO.arDI[78]/Ch[12] <-> Module 6 (GL20-1600END)/1600END input-bit maping/Digital input CH2-bit4
//     PlcTask Inputs/G_IO.arDI[78]/Ch[13] <-> Module 6 (GL20-1600END)/1600END input-bit maping/Digital input CH2-bit5
//     PlcTask Inputs/G_IO.arDI[78]/Ch[14] <-> Module 6 (GL20-1600END)/1600END input-bit maping/Digital input CH2-bit6
//     PlcTask Inputs/G_IO.arDI[78]/Ch[15] <-> Module 6 (GL20-1600END)/1600END input-bit maping/Digital input CH2-bit7
//     PlcTask Inputs/G_IO.arDI[78]/Ch[1] <-> Module 6 (GL20-1600END)/1600END input-bit maping/Digital input CH1-bit1
//     PlcTask Inputs/G_IO.arDI[78]/Ch[2] <-> Module 6 (GL20-1600END)/1600END input-bit maping/Digital input CH1-bit2
//     PlcTask Inputs/G_IO.arDI[78]/Ch[3] <-> Module 6 (GL20-1600END)/1600END input-bit maping/Digital input CH1-bit3
//     PlcTask Inputs/G_IO.arDI[78]/Ch[4] <-> Module 6 (GL20-1600END)/1600END input-bit maping/Digital input CH1-bit4
//     PlcTask Inputs/G_IO.arDI[78]/Ch[5] <-> Module 6 (GL20-1600END)/1600END input-bit maping/Digital input CH1-bit5
//     PlcTask Inputs/G_IO.arDI[78]/Ch[6] <-> Module 6 (GL20-1600END)/1600END input-bit maping/Digital input CH1-bit6
//     PlcTask Inputs/G_IO.arDI[78]/Ch[7] <-> Module 6 (GL20-1600END)/1600END input-bit maping/Digital input CH1-bit7
//     PlcTask Inputs/G_IO.arDI[78]/Ch[8] <-> Module 6 (GL20-1600END)/1600END input-bit maping/Digital input CH2-bit0
//     PlcTask Inputs/G_IO.arDI[78]/Ch[9] <-> Module 6 (GL20-1600END)/1600END input-bit maping/Digital input CH2-bit1
//     PlcTask Outputs/G_IO.arDO[58]/Ch[0] <-> Module 7 (GL20-0016ETP)/0016ETP Output-bit maping/Digital output CH1-bit0
//     PlcTask Outputs/G_IO.arDO[58]/Ch[10] <-> Module 7 (GL20-0016ETP)/0016ETP Output-bit maping/Digital output CH2-bit2
//     PlcTask Outputs/G_IO.arDO[58]/Ch[11] <-> Module 7 (GL20-0016ETP)/0016ETP Output-bit maping/Digital output CH2-bit3
//     PlcTask Outputs/G_IO.arDO[58]/Ch[12] <-> Module 7 (GL20-0016ETP)/0016ETP Output-bit maping/Digital output CH2-bit4
//     PlcTask Outputs/G_IO.arDO[58]/Ch[13] <-> Module 7 (GL20-0016ETP)/0016ETP Output-bit maping/Digital output CH2-bit5
//     PlcTask Outputs/G_IO.arDO[58]/Ch[14] <-> Module 7 (GL20-0016ETP)/0016ETP Output-bit maping/Digital output CH2-bit6
//     PlcTask Outputs/G_IO.arDO[58]/Ch[15] <-> Module 7 (GL20-0016ETP)/0016ETP Output-bit maping/Digital output CH2-bit7
//     PlcTask Outputs/G_IO.arDO[58]/Ch[1] <-> Module 7 (GL20-0016ETP)/0016ETP Output-bit maping/Digital output CH1-bit1
//     PlcTask Outputs/G_IO.arDO[58]/Ch[2] <-> Module 7 (GL20-0016ETP)/0016ETP Output-bit maping/Digital output CH1-bit2
//     PlcTask Outputs/G_IO.arDO[58]/Ch[3] <-> Module 7 (GL20-0016ETP)/0016ETP Output-bit maping/Digital output CH1-bit3
//     PlcTask Outputs/G_IO.arDO[58]/Ch[4] <-> Module 7 (GL20-0016ETP)/0016ETP Output-bit maping/Digital output CH1-bit4
//     PlcTask Outputs/G_IO.arDO[58]/Ch[5] <-> Module 7 (GL20-0016ETP)/0016ETP Output-bit maping/Digital output CH1-bit5
//     PlcTask Outputs/G_IO.arDO[58]/Ch[6] <-> Module 7 (GL20-0016ETP)/0016ETP Output-bit maping/Digital output CH1-bit6
//     PlcTask Outputs/G_IO.arDO[58]/Ch[7] <-> Module 7 (GL20-0016ETP)/0016ETP Output-bit maping/Digital output CH1-bit7
//     PlcTask Outputs/G_IO.arDO[58]/Ch[8] <-> Module 7 (GL20-0016ETP)/0016ETP Output-bit maping/Digital output CH2-bit0
//     PlcTask Outputs/G_IO.arDO[58]/Ch[9] <-> Module 7 (GL20-0016ETP)/0016ETP Output-bit maping/Digital output CH2-bit1
//     PlcTask Outputs/G_IO.arDO[59]/Ch[0] <-> Module 8 (GL20-0016ETP)/0016ETP Output-bit maping/Digital output CH1-bit0
//     PlcTask Outputs/G_IO.arDO[59]/Ch[10] <-> Module 8 (GL20-0016ETP)/0016ETP Output-bit maping/Digital output CH2-bit2
//     PlcTask Outputs/G_IO.arDO[59]/Ch[11] <-> Module 8 (GL20-0016ETP)/0016ETP Output-bit maping/Digital output CH2-bit3
//     PlcTask Outputs/G_IO.arDO[59]/Ch[12] <-> Module 8 (GL20-0016ETP)/0016ETP Output-bit maping/Digital output CH2-bit4
//     PlcTask Outputs/G_IO.arDO[59]/Ch[13] <-> Module 8 (GL20-0016ETP)/0016ETP Output-bit maping/Digital output CH2-bit5
//     PlcTask Outputs/G_IO.arDO[59]/Ch[14] <-> Module 8 (GL20-0016ETP)/0016ETP Output-bit maping/Digital output CH2-bit6
//     PlcTask Outputs/G_IO.arDO[59]/Ch[15] <-> Module 8 (GL20-0016ETP)/0016ETP Output-bit maping/Digital output CH2-bit7
//     PlcTask Outputs/G_IO.arDO[59]/Ch[1] <-> Module 8 (GL20-0016ETP)/0016ETP Output-bit maping/Digital output CH1-bit1
//     PlcTask Outputs/G_IO.arDO[59]/Ch[2] <-> Module 8 (GL20-0016ETP)/0016ETP Output-bit maping/Digital output CH1-bit2
//     PlcTask Outputs/G_IO.arDO[59]/Ch[3] <-> Module 8 (GL20-0016ETP)/0016ETP Output-bit maping/Digital output CH1-bit3
//     PlcTask Outputs/G_IO.arDO[59]/Ch[4] <-> Module 8 (GL20-0016ETP)/0016ETP Output-bit maping/Digital output CH1-bit4
//     PlcTask Outputs/G_IO.arDO[59]/Ch[5] <-> Module 8 (GL20-0016ETP)/0016ETP Output-bit maping/Digital output CH1-bit5
//     PlcTask Outputs/G_IO.arDO[59]/Ch[6] <-> Module 8 (GL20-0016ETP)/0016ETP Output-bit maping/Digital output CH1-bit6
//     PlcTask Outputs/G_IO.arDO[59]/Ch[7] <-> Module 8 (GL20-0016ETP)/0016ETP Output-bit maping/Digital output CH1-bit7
//     PlcTask Outputs/G_IO.arDO[59]/Ch[8] <-> Module 8 (GL20-0016ETP)/0016ETP Output-bit maping/Digital output CH2-bit0
//     PlcTask Outputs/G_IO.arDO[59]/Ch[9] <-> Module 8 (GL20-0016ETP)/0016ETP Output-bit maping/Digital output CH2-bit1
//   kittingDeca/kittingDeca Instance <-> pm side/pm4_5_innerConv
//     PlcTask Inputs/GVL.pm[4].inConv.belt[0].fbconverter.running_freq <-> Axis#1 Iutputs/Axis1 Running frequency
//     PlcTask Inputs/GVL.pm[4].inConv.belt[1].fbconverter.running_freq <-> Axis#2 Iutputs/Axis2 Running frequency
//     PlcTask Inputs/GVL.pm[4].inConv.belt[2].fbconverter.running_freq <-> Axis#3 Iutputs/Axis3 Running frequency
//     PlcTask Inputs/GVL.pm[5].inConv.belt[0].fbconverter.running_freq <-> Axis#4 Iutputs/Axis4 Running frequency
//     PlcTask Inputs/GVL.pm[5].inConv.belt[1].fbconverter.running_freq <-> Axis#5 Iutputs/Axis5 Running frequency
//     PlcTask Inputs/GVL.pm[5].inConv.belt[2].fbconverter.running_freq <-> Axis#6 Iutputs/Axis6 Running frequency
//     PlcTask Inputs/GVL.pm[4].inConv.belt[0].fbconverter.status <-> Axis#1 Iutputs/Axis1 AC drive running status word 2
//     PlcTask Inputs/GVL.pm[4].inConv.belt[1].fbconverter.status <-> Axis#2 Iutputs/Axis2 AC drive running status word 2
//     PlcTask Inputs/GVL.pm[4].inConv.belt[2].fbconverter.status <-> Axis#3 Iutputs/Axis3 AC drive running status word 2
//     PlcTask Inputs/GVL.pm[5].inConv.belt[0].fbconverter.status <-> Axis#4 Iutputs/Axis4 AC drive running status word 2
//     PlcTask Inputs/GVL.pm[5].inConv.belt[1].fbconverter.status <-> Axis#5 Iutputs/Axis5 AC drive running status word 2
//     PlcTask Inputs/GVL.pm[5].inConv.belt[2].fbconverter.status <-> Axis#6 Iutputs/Axis6 AC drive running status word 2
//     PlcTask Outputs/GVL.pm[4].inConv.belt[0].fbconverter.cmd <-> Axis#1 Outputs/Axis1 Communication control command
//     PlcTask Outputs/GVL.pm[4].inConv.belt[1].fbconverter.cmd <-> Axis#2 Outputs/Axis2 Communication control command
//     PlcTask Outputs/GVL.pm[4].inConv.belt[2].fbconverter.cmd <-> Axis#3 Outputs/Axis3 Communication control command
//     PlcTask Outputs/GVL.pm[5].inConv.belt[0].fbconverter.cmd <-> Axis#4 Outputs/Axis4 Communication control command
//     PlcTask Outputs/GVL.pm[5].inConv.belt[1].fbconverter.cmd <-> Axis#5 Outputs/Axis5 Communication control command
//     PlcTask Outputs/GVL.pm[5].inConv.belt[2].fbconverter.cmd <-> Axis#6 Outputs/Axis6 Communication control command
//     PlcTask Outputs/GVL.pm[4].inConv.belt[0].fbconverter.freq <-> Axis#1 Outputs/Axis1 Frequency set through communication
//     PlcTask Outputs/GVL.pm[4].inConv.belt[1].fbconverter.freq <-> Axis#2 Outputs/Axis2 Frequency set through communication
//     PlcTask Outputs/GVL.pm[4].inConv.belt[2].fbconverter.freq <-> Axis#3 Outputs/Axis3 Frequency set through communication
//     PlcTask Outputs/GVL.pm[5].inConv.belt[0].fbconverter.freq <-> Axis#4 Outputs/Axis4 Frequency set through communication
//     PlcTask Outputs/GVL.pm[5].inConv.belt[1].fbconverter.freq <-> Axis#5 Outputs/Axis5 Frequency set through communication
//     PlcTask Outputs/GVL.pm[5].inConv.belt[2].fbconverter.freq <-> Axis#6 Outputs/Axis6 Frequency set through communication
//   kittingDeca/kittingDeca Instance <-> pm side/pm4_5_outerConv
//     PlcTask Inputs/GVL.pm[4].outConv.belt[0].fbconverter.running_freq <-> Axis#1 Iutputs/Axis1 Running frequency
//     PlcTask Inputs/GVL.pm[4].outConv.belt[1].fbconverter.running_freq <-> Axis#2 Iutputs/Axis2 Running frequency
//     PlcTask Inputs/GVL.pm[5].outConv.belt[0].fbconverter.running_freq <-> Axis#3 Iutputs/Axis3 Running frequency
//     PlcTask Inputs/GVL.pm[5].outConv.belt[1].fbconverter.running_freq <-> Axis#4 Iutputs/Axis4 Running frequency
//     PlcTask Inputs/GVL.pm[4].outConv.belt[0].fbconverter.status <-> Axis#1 Iutputs/Axis1 AC drive running status word 2
//     PlcTask Inputs/GVL.pm[4].outConv.belt[1].fbconverter.status <-> Axis#2 Iutputs/Axis2 AC drive running status word 2
//     PlcTask Inputs/GVL.pm[5].outConv.belt[0].fbconverter.status <-> Axis#3 Iutputs/Axis3 AC drive running status word 2
//     PlcTask Inputs/GVL.pm[5].outConv.belt[1].fbconverter.status <-> Axis#4 Iutputs/Axis4 AC drive running status word 2
//     PlcTask Outputs/GVL.pm[4].outConv.belt[0].fbconverter.cmd <-> Axis#1 Outputs/Axis1 Communication control command
//     PlcTask Outputs/GVL.pm[4].outConv.belt[1].fbconverter.cmd <-> Axis#2 Outputs/Axis2 Communication control command
//     PlcTask Outputs/GVL.pm[5].outConv.belt[0].fbconverter.cmd <-> Axis#3 Outputs/Axis3 Communication control command
//     PlcTask Outputs/GVL.pm[5].outConv.belt[1].fbconverter.cmd <-> Axis#4 Outputs/Axis4 Communication control command
//     PlcTask Outputs/GVL.pm[4].outConv.belt[0].fbconverter.freq <-> Axis#1 Outputs/Axis1 Frequency set through communication
//     PlcTask Outputs/GVL.pm[4].outConv.belt[1].fbconverter.freq <-> Axis#2 Outputs/Axis2 Frequency set through communication
//     PlcTask Outputs/GVL.pm[5].outConv.belt[0].fbconverter.freq <-> Axis#3 Outputs/Axis3 Frequency set through communication
//     PlcTask Outputs/GVL.pm[5].outConv.belt[1].fbconverter.freq <-> Axis#4 Outputs/Axis4 Frequency set through communication
//   kittingDeca/kittingDeca Instance <-> pm side/pm6_7_dio
//     PlcTask Inputs/G_IO.arDI[65]/Ch[0] <-> Module 1 (GL20-1600END)/1600END input-bit maping/Digital input CH1-bit0
//     PlcTask Inputs/G_IO.arDI[65]/Ch[10] <-> Module 1 (GL20-1600END)/1600END input-bit maping/Digital input CH2-bit2
//     PlcTask Inputs/G_IO.arDI[65]/Ch[11] <-> Module 1 (GL20-1600END)/1600END input-bit maping/Digital input CH2-bit3
//     PlcTask Inputs/G_IO.arDI[65]/Ch[12] <-> Module 1 (GL20-1600END)/1600END input-bit maping/Digital input CH2-bit4
//     PlcTask Inputs/G_IO.arDI[65]/Ch[13] <-> Module 1 (GL20-1600END)/1600END input-bit maping/Digital input CH2-bit5
//     PlcTask Inputs/G_IO.arDI[65]/Ch[14] <-> Module 1 (GL20-1600END)/1600END input-bit maping/Digital input CH2-bit6
//     PlcTask Inputs/G_IO.arDI[65]/Ch[15] <-> Module 1 (GL20-1600END)/1600END input-bit maping/Digital input CH2-bit7
//     PlcTask Inputs/G_IO.arDI[65]/Ch[1] <-> Module 1 (GL20-1600END)/1600END input-bit maping/Digital input CH1-bit1
//     PlcTask Inputs/G_IO.arDI[65]/Ch[2] <-> Module 1 (GL20-1600END)/1600END input-bit maping/Digital input CH1-bit2
//     PlcTask Inputs/G_IO.arDI[65]/Ch[3] <-> Module 1 (GL20-1600END)/1600END input-bit maping/Digital input CH1-bit3
//     PlcTask Inputs/G_IO.arDI[65]/Ch[4] <-> Module 1 (GL20-1600END)/1600END input-bit maping/Digital input CH1-bit4
//     PlcTask Inputs/G_IO.arDI[65]/Ch[5] <-> Module 1 (GL20-1600END)/1600END input-bit maping/Digital input CH1-bit5
//     PlcTask Inputs/G_IO.arDI[65]/Ch[6] <-> Module 1 (GL20-1600END)/1600END input-bit maping/Digital input CH1-bit6
//     PlcTask Inputs/G_IO.arDI[65]/Ch[7] <-> Module 1 (GL20-1600END)/1600END input-bit maping/Digital input CH1-bit7
//     PlcTask Inputs/G_IO.arDI[65]/Ch[8] <-> Module 1 (GL20-1600END)/1600END input-bit maping/Digital input CH2-bit0
//     PlcTask Inputs/G_IO.arDI[65]/Ch[9] <-> Module 1 (GL20-1600END)/1600END input-bit maping/Digital input CH2-bit1
//     PlcTask Inputs/G_IO.arDI[66]/Ch[0] <-> Module 2 (GL20-1600END)/1600END input-bit maping/Digital input CH1-bit0
//     PlcTask Inputs/G_IO.arDI[66]/Ch[10] <-> Module 2 (GL20-1600END)/1600END input-bit maping/Digital input CH2-bit2
//     PlcTask Inputs/G_IO.arDI[66]/Ch[11] <-> Module 2 (GL20-1600END)/1600END input-bit maping/Digital input CH2-bit3
//     PlcTask Inputs/G_IO.arDI[66]/Ch[12] <-> Module 2 (GL20-1600END)/1600END input-bit maping/Digital input CH2-bit4
//     PlcTask Inputs/G_IO.arDI[66]/Ch[13] <-> Module 2 (GL20-1600END)/1600END input-bit maping/Digital input CH2-bit5
//     PlcTask Inputs/G_IO.arDI[66]/Ch[14] <-> Module 2 (GL20-1600END)/1600END input-bit maping/Digital input CH2-bit6
//     PlcTask Inputs/G_IO.arDI[66]/Ch[15] <-> Module 2 (GL20-1600END)/1600END input-bit maping/Digital input CH2-bit7
//     PlcTask Inputs/G_IO.arDI[66]/Ch[1] <-> Module 2 (GL20-1600END)/1600END input-bit maping/Digital input CH1-bit1
//     PlcTask Inputs/G_IO.arDI[66]/Ch[2] <-> Module 2 (GL20-1600END)/1600END input-bit maping/Digital input CH1-bit2
//     PlcTask Inputs/G_IO.arDI[66]/Ch[3] <-> Module 2 (GL20-1600END)/1600END input-bit maping/Digital input CH1-bit3
//     PlcTask Inputs/G_IO.arDI[66]/Ch[4] <-> Module 2 (GL20-1600END)/1600END input-bit maping/Digital input CH1-bit4
//     PlcTask Inputs/G_IO.arDI[66]/Ch[5] <-> Module 2 (GL20-1600END)/1600END input-bit maping/Digital input CH1-bit5
//     PlcTask Inputs/G_IO.arDI[66]/Ch[6] <-> Module 2 (GL20-1600END)/1600END input-bit maping/Digital input CH1-bit6
//     PlcTask Inputs/G_IO.arDI[66]/Ch[7] <-> Module 2 (GL20-1600END)/1600END input-bit maping/Digital input CH1-bit7
//     PlcTask Inputs/G_IO.arDI[66]/Ch[8] <-> Module 2 (GL20-1600END)/1600END input-bit maping/Digital input CH2-bit0
//     PlcTask Inputs/G_IO.arDI[66]/Ch[9] <-> Module 2 (GL20-1600END)/1600END input-bit maping/Digital input CH2-bit1
//     PlcTask Inputs/G_IO.arDI[67]/Ch[0] <-> Module 3 (GL20-1600END)/1600END input-bit maping/Digital input CH1-bit0
//     PlcTask Inputs/G_IO.arDI[67]/Ch[10] <-> Module 3 (GL20-1600END)/1600END input-bit maping/Digital input CH2-bit2
//     PlcTask Inputs/G_IO.arDI[67]/Ch[11] <-> Module 3 (GL20-1600END)/1600END input-bit maping/Digital input CH2-bit3
//     PlcTask Inputs/G_IO.arDI[67]/Ch[12] <-> Module 3 (GL20-1600END)/1600END input-bit maping/Digital input CH2-bit4
//     PlcTask Inputs/G_IO.arDI[67]/Ch[13] <-> Module 3 (GL20-1600END)/1600END input-bit maping/Digital input CH2-bit5
//     PlcTask Inputs/G_IO.arDI[67]/Ch[14] <-> Module 3 (GL20-1600END)/1600END input-bit maping/Digital input CH2-bit6
//     PlcTask Inputs/G_IO.arDI[67]/Ch[15] <-> Module 3 (GL20-1600END)/1600END input-bit maping/Digital input CH2-bit7
//     PlcTask Inputs/G_IO.arDI[67]/Ch[1] <-> Module 3 (GL20-1600END)/1600END input-bit maping/Digital input CH1-bit1
//     PlcTask Inputs/G_IO.arDI[67]/Ch[2] <-> Module 3 (GL20-1600END)/1600END input-bit maping/Digital input CH1-bit2
//     PlcTask Inputs/G_IO.arDI[67]/Ch[3] <-> Module 3 (GL20-1600END)/1600END input-bit maping/Digital input CH1-bit3
//     PlcTask Inputs/G_IO.arDI[67]/Ch[4] <-> Module 3 (GL20-1600END)/1600END input-bit maping/Digital input CH1-bit4
//     PlcTask Inputs/G_IO.arDI[67]/Ch[5] <-> Module 3 (GL20-1600END)/1600END input-bit maping/Digital input CH1-bit5
//     PlcTask Inputs/G_IO.arDI[67]/Ch[6] <-> Module 3 (GL20-1600END)/1600END input-bit maping/Digital input CH1-bit6
//     PlcTask Inputs/G_IO.arDI[67]/Ch[7] <-> Module 3 (GL20-1600END)/1600END input-bit maping/Digital input CH1-bit7
//     PlcTask Inputs/G_IO.arDI[67]/Ch[8] <-> Module 3 (GL20-1600END)/1600END input-bit maping/Digital input CH2-bit0
//     PlcTask Inputs/G_IO.arDI[67]/Ch[9] <-> Module 3 (GL20-1600END)/1600END input-bit maping/Digital input CH2-bit1
//     PlcTask Inputs/G_IO.arDI[68]/Ch[0] <-> Module 4 (GL20-1600END)/1600END input-bit maping/Digital input CH1-bit0
//     PlcTask Inputs/G_IO.arDI[68]/Ch[10] <-> Module 4 (GL20-1600END)/1600END input-bit maping/Digital input CH2-bit2
//     PlcTask Inputs/G_IO.arDI[68]/Ch[11] <-> Module 4 (GL20-1600END)/1600END input-bit maping/Digital input CH2-bit3
//     PlcTask Inputs/G_IO.arDI[68]/Ch[12] <-> Module 4 (GL20-1600END)/1600END input-bit maping/Digital input CH2-bit4
//     PlcTask Inputs/G_IO.arDI[68]/Ch[13] <-> Module 4 (GL20-1600END)/1600END input-bit maping/Digital input CH2-bit5
//     PlcTask Inputs/G_IO.arDI[68]/Ch[14] <-> Module 4 (GL20-1600END)/1600END input-bit maping/Digital input CH2-bit6
